// TIA Portal V19 program export: 1 tag tables, 0 data types, 14 data blocks, 15 code blocks (in call order from the OBs), 30 instance data blocks

VAR_GLOBAL   // PLC tag table "Default tag table"
   "EMG STOP" AT %I0.0 : Bool;
   "HOOTER RESET" AT %I0.1 : Bool;
   "PHASE FAIL" AT %I0.2 : Bool;
   "AIR PRESSURE FAIL" AT %I0.3 : Bool;
   "SYRUP MFG VESSEL BOTTOM STERROR TRIP" AT %I0.4 : Bool;
   "PREMIXING VESSEL BOTTOM STERROR TRIP" AT %I0.5 : Bool;
   "INLINE 1 HOMOGENIZER MOTOR1 TRIP" AT %I0.6 : Bool;
   "INLINE 2 HOMOGENIZER MOTOR 2 TRIP" AT %I0.7 : Bool;
   "FILTER PRESS MOTOR 1 TRIP" AT %I1.0 : Bool;
   "FILTER PRESS MOTOR 2 TRIP" AT %I1.1 : Bool;
   "VACCUM PUMP MOTOR 1 TRIP" AT %I1.2 : Bool;
   "VACCUMP PUMP MOTOR 2 TRIP" AT %I1.3 : Bool;
   "VACCUMP PUMP MOTOR 3 TRIP" AT %I1.4 : Bool;
   "VACCUMP PUMP MOTOR 4 TRIP" AT %I1.5 : Bool;
   "SUGAR VESSEL BOTTOM STERROR TRIP" AT %I1.6 : Bool;
   "BASKET FILTER MOTOR TRIP" AT %I1.7 : Bool;
   "SYRUP FLOW SWITCH" AT %I2.0 : Bool;
   "PREMIXING FLOW SWITCH" AT %I2.1 : Bool;
   "SUGAR FLOW SWITCH" AT %I2.2 : Bool;
   "INLINE 1 FLOW SWITCH" AT %I2.3 : Bool;
   "INLINE 2 FLOW SWITCH" AT %I2.4 : Bool;
   "HOOTER RESET 2" AT %I2.5 : Bool;
   SPARE_DI1 AT %I2.6 : Bool;
   SPARE_DI2 AT %I2.7 : Bool;
   SPARE_DI3 AT %I3.0 : Bool;
   SPARE_DI4 AT %I3.1 : Bool;
   SPARE_DI5 AT %I3.2 : Bool;
   SPARE_DI6 AT %I3.3 : Bool;
   SPARE_DI7 AT %I3.4 : Bool;
   SPARE_DI8 AT %I3.5 : Bool;
   SPARE_DI9 AT %I3.6 : Bool;
   SPARE_DI10 AT %I3.7 : Bool;
   "SYRUP MFG VESSEL BOTTOM STERROR RUN" AT %Q0.0 : Bool;
   "PREMIXING VESSEL BOTTOM STERROR RUN" AT %Q0.1 : Bool;
   "INLINE 1 HOMOGENIZER MOTOR1 RUN" AT %Q0.2 : Bool;
   "INLINE 2 HOMOGENIZER MOTOR 2 RUN" AT %Q0.3 : Bool;
   "FILTER PRESS MOTOR 1 RUN" AT %Q0.4 : Bool;
   "FILTER PRESS MOTOR 2 RUN" AT %Q0.5 : Bool;
   "VACCUM PUMP MOTOR 1 RUN" AT %Q0.6 : Bool;
   "VACCUMP PUMP MOTOR 2 RUN" AT %Q0.7 : Bool;
   "VACCUMP PUMP MOTOR 3 RUN" AT %Q1.0 : Bool;
   "VACCUMP PUMP MOTOR 4 RUN" AT %Q1.1 : Bool;
   "SUGAR VESSEL BOTTOM STERROR RUN" AT %Q1.2 : Bool;
   "BASKET FILTER MOTOR RUN" AT %Q1.3 : Bool;
   "PBV-01" AT %Q1.4 : Bool;
   "PBV-02" AT %Q1.5 : Bool;
   "PBV-03" AT %Q1.6 : Bool;
   "PBV-04" AT %Q1.7 : Bool;
   "PBV-07" AT %Q2.0 : Bool;
   "PAV-09" AT %Q2.1 : Bool;
   "PAV-10" AT %Q2.2 : Bool;
   "PAV-11" AT %Q2.3 : Bool;
   "PAV-12" AT %Q2.4 : Bool;
   "PAV-13" AT %Q2.5 : Bool;
   "PAV-14" AT %Q2.6 : Bool;
   "PBV-15" AT %Q2.7 : Bool;
   "PBV-16" AT %Q3.0 : Bool;
   "PFBV-17" AT %Q3.1 : Bool;
   "PBV-19" AT %Q3.2 : Bool;
   "PBV-20" AT %Q3.3 : Bool;
   "PBV-21" AT %Q3.4 : Bool;
   "PBV-22" AT %Q3.5 : Bool;
   "PBV-25" AT %Q3.6 : Bool;
   "PBV-27" AT %Q3.7 : Bool;
   "PAV-28" AT %Q4.0 : Bool;
   "PAV-29" AT %Q4.1 : Bool;
   "PBV-30" AT %Q4.2 : Bool;
   "PBV-31" AT %Q4.3 : Bool;
   "PFBV-32" AT %Q4.4 : Bool;
   "PBV-36" AT %Q4.5 : Bool;
   "PBV-37" AT %Q4.6 : Bool;
   "PBV-38" AT %Q4.7 : Bool;
   "PBV-41" AT %Q5.0 : Bool;
   "PAV-50" AT %Q5.1 : Bool;
   "PAV-51" AT %Q5.2 : Bool;
   "PAV-52" AT %Q5.3 : Bool;
   "PAV-53" AT %Q5.4 : Bool;
   "PAV-54" AT %Q5.5 : Bool;
   "PAV-55" AT %Q5.6 : Bool;
   "PAV-56" AT %Q5.7 : Bool;
   "PBV-57" AT %Q6.0 : Bool;
   "PFBV-59" AT %Q6.1 : Bool;
   "PBV-79" AT %Q6.2 : Bool;
   "PBV-80" AT %Q6.3 : Bool;
   "PBV-81" AT %Q6.4 : Bool;
   "PBV-82" AT %Q6.5 : Bool;
   "PBV-83" AT %Q6.6 : Bool;
   "PBV-84" AT %Q6.7 : Bool;
   "PBV-85" AT %Q7.0 : Bool;
   "PBV-86" AT %Q7.1 : Bool;
   "PBV-87" AT %Q7.2 : Bool;
   "PBV-88" AT %Q7.3 : Bool;
   "PBV-89" AT %Q7.4 : Bool;
   "PBV-90" AT %Q7.5 : Bool;
   "PBV-91" AT %Q7.6 : Bool;
   "PBV-92" AT %Q7.7 : Bool;
   "PBV-93" AT %Q8.0 : Bool;
   "PBV-94" AT %Q8.1 : Bool;
   "PBV-95" AT %Q8.2 : Bool;
   "PBV-96" AT %Q8.3 : Bool;
   "PBV-97" AT %Q8.4 : Bool;
   "PBV-98" AT %Q8.5 : Bool;
   "PAV-99" AT %Q8.6 : Bool;
   "PBV-100" AT %Q8.7 : Bool;
   "PBV-101" AT %Q9.0 : Bool;
   "PBV-102" AT %Q9.1 : Bool;
   "PBV-103" AT %Q9.2 : Bool;
   "PBV-104" AT %Q9.3 : Bool;
   "PBV-105" AT %Q9.4 : Bool;
   "PBV-106" AT %Q9.5 : Bool;
   "PBV-107" AT %Q9.6 : Bool;
   "PBV-108" AT %Q9.7 : Bool;
   "PBV-109" AT %Q10.0 : Bool;
   "PBV-110" AT %Q10.1 : Bool;
   "PBV-111" AT %Q10.2 : Bool;
   "PBV-112" AT %Q10.3 : Bool;
   "PAV-113" AT %Q10.4 : Bool;
   "PBV-114" AT %Q10.5 : Bool;
   "PBV-115" AT %Q10.6 : Bool;
   "PBV-116" AT %Q10.7 : Bool;
   "PBV-117" AT %Q11.0 : Bool;
   "PBV-118" AT %Q11.1 : Bool;
   "PBV-119" AT %Q11.2 : Bool;
   "PBV-120" AT %Q11.3 : Bool;
   "PBV-121" AT %Q11.4 : Bool;
   "PBV-122" AT %Q11.5 : Bool;
   "PBV-123" AT %Q11.6 : Bool;
   "PBV-124" AT %Q11.7 : Bool;
   "PBV-149" AT %Q12.0 : Bool;
   "PBV-150" AT %Q12.1 : Bool;
   "PBV-151" AT %Q12.2 : Bool;
   "PBV-152" AT %Q12.3 : Bool;
   "PBV-153" AT %Q12.4 : Bool;
   "PBV-155" AT %Q12.5 : Bool;
   "PBV-156" AT %Q12.6 : Bool;
   HOOTER_1 AT %Q12.7 : Bool;
   HOOTR_2 AT %Q13.0 : Bool;
   SPARE_DO1 AT %Q13.1 : Bool;
   SPARE_DO2 AT %Q13.2 : Bool;
   SPARE_DO3 AT %Q13.3 : Bool;
   SPARE_DO4 AT %Q13.4 : Bool;
   SPARE_DO5 AT %Q13.5 : Bool;
   SPARE_DO6 AT %Q13.6 : Bool;
   SPARE_DO7 AT %Q13.7 : Bool;
   SPARE_8 AT %Q23.0 : Bool;
   SPARE_9 AT %Q23.1 : Bool;
   SPARE_10 AT %Q23.2 : Bool;
   SPARE_11 AT %Q23.3 : Bool;
   SPARE_12 AT %Q23.4 : Bool;
   SPARE_13 AT %Q23.5 : Bool;
   SPARE_14 AT %Q23.6 : Bool;
   SPARE_15 AT %Q23.7 : Bool;
   SPARE_16 AT %Q24.0 : Bool;
   SPARE_17 AT %Q24.1 : Bool;
   SPARE_18 AT %Q24.2 : Bool;
   SPARE_19 AT %Q24.3 : Bool;
   SPARE_20 AT %Q24.4 : Bool;
   SPARE_21 AT %Q24.5 : Bool;
   SPARE_22 AT %Q24.6 : Bool;
   SPARE_23 AT %Q24.7 : Bool;
   "SYRUP VESSEL TEMP SENSOR" AT %IW4 : Int;
   "PREMIXING VESSEL TEMP SENSOR" AT %IW6 : Int;
   "SUGAR VESSEL TEMP SENSOR" AT %IW8 : Int;
   "STEAM LINE_1 TEMP SENSOR" AT %IW10 : Int;
   "STEAM LINE_2 TEMP SENSOR" AT %IW12 : Int;
   "PRESSURE TRANSMITTER 1" AT %IW14 : Int;
   "PRESSURE TRANSMITTER 2" AT %IW16 : Int;
   "VACCIM TRANSMITTER 1" AT %IW18 : Int;
   "VACCIM TRANSMITTER 2" AT %IW20 : Int;
   "VACCUM TRANSMITTER 3" AT %IW22 : Int;
   "SYRUP LOAD CELL" AT %IW24 : Int;
   "PREMIXING LOAD CELL" AT %IW26 : Int;
   "SUGAR LOAD CELL" AT %IW28 : Int;
   "ULTRASONIC LEVEL SENSOR-1" AT %IW30 : Int;
   "ULTRASONIC LEVEL SENSOR-2" AT %IW32 : Int;
   "ULTRASONIC LEVEL SENSOR-3" AT %IW34 : Int;
   "SYRUP MFG VESSEL SPEED" AT %QW15 : Int;
   "PREMIXING VESSEL SPEED" AT %QW17 : Int;
   "SUGAR VESSEL SPEED" AT %QW19 : Int;
   "SPARE(17)" AT %QW21 : Int;
   System_Byte AT %MB1 : Byte;
   DiagStatusUpdate AT %M1.1 : Bool;
   AlwaysTRUE AT %M1.2 : Bool;
   AlwaysFALSE AT %M1.3 : Bool;
   Clock_Byte AT %MB0 : Byte;
   Clock_10Hz AT %M0.0 : Bool;
   Clock_5Hz AT %M0.1 : Bool;
   "Clock_2.5Hz" AT %M0.2 : Bool;
   Clock_2Hz AT %M0.3 : Bool;
   "Clock_1.25Hz" AT %M0.4 : Bool;
   Clock_1Hz AT %M0.5 : Bool;
   "Clock_0.625Hz" AT %M0.6 : Bool;
   "Clock_0.5Hz" AT %M0.7 : Bool;
   "Vaccup Pump2-W bit" AT %M6.0 : Bool;
   "Vaccup Pump2-S bit" AT %M6.1 : Bool;
   YY AT %M4.0 : Bool;
   "MFG LOVE CALCULATE PV" AT %MD8 : Real;
   hh1 AT %MD12 : Real;
   "MFG MOVE PV LOAD CELL" AT %MD16 : Real;
   LL AT %M2.0 : Bool;
END_VAR

DATA_BLOCK "DI MAPING"   // DB1
{ S7_Optimized_Access := 'FALSE' }
   VAR
      "EMG STOP" : Bool;
      "HOOTER RESET_1" : Bool;
      "PHASE FAIL" : Bool;
      "AIR PRESSURE FAIL" : Bool;
      "SYRUP MFG VESSEL BOTTOM STERROR TRIP" : Bool;
      "PREMIXING VESSEL BOTTOM STERROR TRIP" : Bool;
      "INLINE 1 HOMOGENIZER MOTOR1 TRIP" : Bool;
      "INLINE 2 HOMOGENIZER MOTOR 2 TRIP" : Bool;
      "FILTER PRESS MOTOR 1 TRIP" : Bool;
      "FILTER PRESS MOTOR 2 TRIP" : Bool;
      "VACCUM PUMP MOTOR 1 TRIP" : Bool;
      "VACCUMP PUMP MOTOR 2 TRIP" : Bool;
      "VACCUMP PUMP MOTOR 3 TRIP" : Bool;
      "VACCUMP PUMP MOTOR 4 TRIP" : Bool;
      "SUGAR VESSEL BOTTOM STERROR TRIP" : Bool;
      "BASKET FILTER MOTOR TRIP" : Bool;
      "SYRUP FLOW SWITCH" : Bool;
      "PREMIXING FLOW SWITCH" : Bool;
      "SUGAR FLOW SWITCH" : Bool;
      "INLINE 1 FLOW SWITCH" : Bool;
      "INLINE 2 FLOW SWITCH" : Bool;
      "HOOTER RESET_2" : Bool;
      SPARE_DI1 : Bool;
      SPARE_DI2 : Bool;
      SPARE_DI3 : Bool;
      SPARE_DI4 : Bool;
      SPARE_DI5 : Bool;
      SPARE_DI6 : Bool;
      SPARE_DI7 : Bool;
      SPARE_DI8 : Bool;
      SPARE_DI9 : Bool;
      SPARE_DI10 : Bool;
   END_VAR
BEGIN
END_DATA_BLOCK

DATA_BLOCK "AUTO SUBOUTPUT DB"   // DB46
{ S7_Optimized_Access := 'TRUE' }
// stored: MemoryReserve 100
   VAR
      "SYRUP MFG VESSEL BOTTOM STERROR RUN" : Bool;
      "PREMIXING VESSEL BOTTOM STERROR RUN" : Bool;
      "INLINE 1 HOMOGENIZER MOTOR1 RUN" : Bool;
      "INLINE 2 HOMOGENIZER MOTOR 2 RUN" : Bool;
      "FILTER PRESS MOTOR 1 RUN" : Bool;
      "FILTER PRESS MOTOR 2 RUN" : Bool;
      "VACCUM PUMP MOTOR-W 1 RUN" : Bool;
      "VACCUMP PUMP MOTOR-S2 RUN" : Bool;
      "VACCUMP PUMP MOTOR-W 3 RUN" : Bool;
      "VACCUMP PUMP MOTOR-S 4 RUN" : Bool;
      "SUGAR VESSEL BOTTOM STERROR RUN" : Bool;
      "BASKET FILTER MOTOR RUN" : Bool;
      "PBV-01 INGREDIENT INLET" : Bool;
      "PBV-02 CIP INLET (SPRAY BALL)" : Bool;
      "PBV-03 VENT FILTER ISOLATION" : Bool;
      "PBV-04 PW INLET" : Bool;
      "PBV-07 PREMIX TANK DRAIN VALVE" : Bool;
      "PAV-09 JACKET STEAM INLET" : Bool;
      "PAV-10 JACKET CONDENSATE DRAIN" : Bool;
      "PAV-11 JACKET BYPASS DRAIN VALVE" : Bool;
      "PAV-12 SEAL COOLING INLET" : Bool;
      "PAV-13 WATER COOLING INLET" : Bool;
      "PAV-14 WATER COOLING OUTLET" : Bool;
      "PBV-15 VACUUM INLET" : Bool;
      "PBV-16 VACUUM VENT VALVE" : Bool;
      "PFBV-17 TANK OUTLET VALVE" : Bool;
      "PBV-19 PW INLET" : Bool;
      "PBV-20 CIP INLET (SPRAY BALL)" : Bool;
      "PBV-21 VENT FILTER ISOLATION" : Bool;
      "PBV-22 INGREDIENT INLET (SUGAR INLET)" : Bool;
      "PBV-25 BOTTOM OUTLET TO DRAIN VALVE" : Bool;
      "PAV-27 JACKET STEAM INLET" : Bool;
      "PAV-28 SEAL COOLING INLET" : Bool;
      "PAV-29 JACKET CONDENSATE DRAIN" : Bool;
      "PBV-30 VACUUM INLET VALVE" : Bool;
      "PBV-31 VACUUM VENT VALVE" : Bool;
      "PFBV-32 TANK OUTLET VALVE" : Bool;
      "PBV-36 PW INLET" : Bool;
      "PBV-37 VENT FILTER ISOLATION" : Bool;
      "PBV-38 CIP INLET LINE" : Bool;
      "PBV-41 MFG TANK DRAIN VALVE" : Bool;
      "PAV-50 JACKET STEAM INLET" : Bool;
      "PAV-51 WATER COOLING OUTLET" : Bool;
      "PAV-52 WATER COOLING INLET" : Bool;
      "PAV-53 SEAL COOLING INLET" : Bool;
      "PAV-54 JACKET STEAM OUTLET VALVE" : Bool;
      "PAV-55 JACKET CONDENSATE BYPASS DRAIN" : Bool;
      "PAV-56 INLINE HOMO. SEAL COOLING INLET" : Bool;
      "PBV-57 VACUUM INLET VALVE" : Bool;
      "PFBV-59 TANK OUTLET VALVE" : Bool;
      "PBV-79 BASKET FILTER INLET" : Bool;
      "PBV-80 BOTTOM OUTLET TO BASKET FILTER" : Bool;
      "PBV-81 TANK BOTTOM OUTLET TO CIP OUTLET" : Bool;
      "PBV-82 CIP ISOLATION" : Bool;
      "PBV-83 PREMIX TRANSFER TO MFG VESSEL TRANSFER (TOP DISH)" : Bool;
      "PBV-84 FROM TANK OUTLET TO CIP OUTLET" : Bool;
      "PBV-85 SORBITOL INLET LINE" : Bool;
      "PBV-86 GLUCOSE INLET LINE" : Bool;
      "PBV-87 BASKET FILTER TO PREMIX VESSEL LINE" : Bool;
      "PBV-88 BASKET FILTER TRANSFER LINE" : Bool;
      "PBV-89 BASKET FILTER TO MFG INLET TRANSFER LINE" : Bool;
      "PBV-90 PREMIX TO MFG TRANSFER LINE" : Bool;
      "PBV-91 PREMIX TO MFG TRANSFER LINE" : Bool;
      "PBV-92 PREMIX TO STORAGE – 4 TRANSFER LINE" : Bool;
      "PBV-93 TANK OUTLET TO INLINE HOMOGENIZER LINE" : Bool;
      "PBV-94 INLINE HOMOGENIZER INLET LINE" : Bool;
      "PBV-95 TANK OUTLET TO FILTER PRESS LINE" : Bool;
      "PBV-96 INLINE HOMOGENIZER RECIRCULATION LINE" : Bool;
      "PBV-97 FILTER PRESS OUTLET" : Bool;
      "PBV-98 INLINE HOMOGENIZER TO FILTER PRESS OUTLET LINE" : Bool;
      "PAV-99 INLINE HOMOGENIZER SEAL COOLING" : Bool;
      "PBV-100 FILTER PRESS INLET" : Bool;
      "PBV-101 SUGAR MELTING TO MFG TRANSFER (TOP DISH)" : Bool;
      "PBV-102 PREMIX TO MFG TRANSFER (TOP DISH)" : Bool;
      "PBV-103 CIP INLET (SPRAY BALL)" : Bool;
      "PBV-104 MFG VESSEL TRANSFER LINE" : Bool;
      "PBV-105 INGREDIENT INLET" : Bool;
      "PBV-106 SORBITOL INLET" : Bool;
      "PBV-107 GLUCOSE INLET" : Bool;
      "PBV-108 INLINE HOMOGENIZER TO FILTER PRESS INLET LINE" : Bool;
      "PBV-109 HOMO. RECIRCULATION INLET" : Bool;
      "PBV-110 INLINE HOMOGENIZER TO INLET LINE" : Bool;
      "PBV-111 FILTER PRESS OUTLER VALVE" : Bool;
      "PBV-112 FILTER PRESS TO TRANSFER LINE" : Bool;
      "PAV-113 TANK OUTLET TO CIP DRAIN LINE" : Bool;
      "PBV-114 TANK OUTLET TO INLINE HOMOGENIZER LINE" : Bool;
      "PBV-115 MFG TO STORAGE – 1 TRANSFER LINE" : Bool;
      "PBV-116 MFG TO STORAGE – 2 TRANSFER LINE" : Bool;
      "PBV-117 MFG TO STORAGE – 3 TRANSFER LINE" : Bool;
      "PBV-118 FILTER PRESS INLET" : Bool;
      "PBV-119 SEAL COOLING FOR STORAGE VESSEL - 4" : Bool;
      "PBV-120 SEAL COOLING FOR STORAGE VESSEL - 3" : Bool;
      "PBV-121 SEAL COOLING FOR STORAGE VESSEL - 2" : Bool;
      "PBV-122 SEAL COOLING FOR STORAGE VESSEL - 1" : Bool;
      "PBV-123 VESSEL TOP DISH" : Bool;
      "PBV-124 VESSEL INLET LINE" : Bool;
      "PBV-149" : Bool;
      "PBV-150" : Bool;
      "PBV-151" : Bool;
      "PBV-152" : Bool;
      "PBV-153" : Bool;
      "PBV-155" : Bool;
      "PBV-156" : Bool;
   END_VAR
BEGIN
END_DATA_BLOCK

DATA_BLOCK "MANUAL BIT"   // DB4
{ S7_Optimized_Access := 'TRUE' }
// stored: MemoryReserve 100
   VAR
      "SYRUP MFG VESSEL BOTTOM STERROR RUN" : Bool;
      "PREMIXING VESSEL BOTTOM STERROR RUN" : Bool;
      "INLINE 1 HOMOGENIZER MOTOR1 RUN" : Bool;
      "INLINE 2 HOMOGENIZER MOTOR 2 RUN" : Bool;
      "FILTER PRESS MOTOR 1 RUN" : Bool;
      "FILTER PRESS MOTOR 2 RUN" : Bool;
      "VACCUM PUMP MOTOR-W 1 RUN" : Bool;
      "VACCUMP PUMP MOTOR-S2 RUN" : Bool;
      "VACCUM PUMP MOTOR-W 1 RUN_1" : Bool;
      "VACCUMP PUMP MOTOR-S2 RUN_1" : Bool;
      "VACCUMP PUMP MOTOR-W 3 RUN" : Bool;
      "VACCUMP PUMP MOTOR-S 4 RUN" : Bool;
      "SUGAR VESSEL BOTTOM STERROR RUN" : Bool;
      "BASKET FILTER MOTOR RUN" : Bool;
      "PBV-01 INGREDIENT INLET" : Bool;
      "PBV-02 CIP INLET (SPRAY BALL)" : Bool;
      "PBV-03 VENT FILTER ISOLATION" : Bool;
      "PBV-04 PW INLET" : Bool;
      "PBV-07 PREMIX TANK DRAIN VALVE" : Bool;
      "PAV-09 JACKET STEAM INLET" : Bool;
      "PAV-10 JACKET CONDENSATE DRAIN" : Bool;
      "PAV-11 JACKET BYPASS DRAIN VALVE" : Bool;
      "PAV-12 SEAL COOLING INLET" : Bool;
      "PAV-13 WATER COOLING INLET" : Bool;
      "PAV-14 WATER COOLING OUTLET" : Bool;
      "PBV-15 VACUUM INLET" : Bool;
      "PBV-16 VACUUM VENT VALVE" : Bool;
      "PFBV-17 TANK OUTLET VALVE" : Bool;
      "PBV-19 PW INLET" : Bool;
      "PBV-20 CIP INLET (SPRAY BALL)" : Bool;
      "PBV-21 VENT FILTER ISOLATION" : Bool;
      "PBV-22 INGREDIENT INLET (SUGAR INLET)" : Bool;
      "PBV-25 BOTTOM OUTLET TO DRAIN VALVE" : Bool;
      "PAV-27 JACKET STEAM INLET" : Bool;
      "PAV-28 SEAL COOLING INLET" : Bool;
      "PAV-29 JACKET CONDENSATE DRAIN" : Bool;
      "PBV-30 VACUUM INLET VALVE" : Bool;
      "PBV-31 VACUUM VENT VALVE" : Bool;
      "PFBV-32 TANK OUTLET VALVE" : Bool;
      "PBV-36 PW INLET" : Bool;
      "PBV-37 VENT FILTER ISOLATION" : Bool;
      "PBV-38 CIP INLET LINE" : Bool;
      "PBV-41 MFG TANK DRAIN VALVE" : Bool;
      "PAV-50 JACKET STEAM INLET" : Bool;
      "PAV-51 WATER COOLING OUTLET" : Bool;
      "PAV-52 WATER COOLING INLET" : Bool;
      "PAV-53 SEAL COOLING INLET" : Bool;
      "PAV-54 JACKET STEAM OUTLET VALVE" : Bool;
      "PAV-55 JACKET CONDENSATE BYPASS DRAIN" : Bool;
      "PAV-56 INLINE HOMO. SEAL COOLING INLET" : Bool;
      "PBV-57 VACUUM INLET VALVE" : Bool;
      "PFBV-59 TANK OUTLET VALVE" : Bool;
      "PBV-79 BASKET FILTER INLET" : Bool;
      "PBV-80 BOTTOM OUTLET TO BASKET FILTER" : Bool;
      "PBV-81 TANK BOTTOM OUTLET TO CIP OUTLET" : Bool;
      "PBV-82 CIP ISOLATION" : Bool;
      "PBV-83 PREMIX TRANSFER TO MFG VESSEL TRANSFER (TOP DISH)" : Bool;
      "PBV-84 FROM TANK OUTLET TO CIP OUTLET" : Bool;
      "PBV-85 SORBITOL INLET LINE" : Bool;
      "PBV-86 GLUCOSE INLET LINE" : Bool;
      "PBV-87 BASKET FILTER TO PREMIX VESSEL LINE" : Bool;
      "PBV-88 BASKET FILTER TRANSFER LINE" : Bool;
      "PBV-89 BASKET FILTER TO MFG INLET TRANSFER LINE" : Bool;
      "PBV-90 PREMIX TO MFG TRANSFER LINE" : Bool;
      "PBV-91 PREMIX TO MFG TRANSFER LINE" : Bool;
      "PBV-92 PREMIX TO STORAGE – 4 TRANSFER LINE" : Bool;
      "PBV-93 TANK OUTLET TO INLINE HOMOGENIZER LINE" : Bool;
      "PBV-94 INLINE HOMOGENIZER INLET LINE" : Bool;
      "PBV-95 TANK OUTLET TO FILTER PRESS LINE" : Bool;
      "PBV-96 INLINE HOMOGENIZER RECIRCULATION LINE" : Bool;
      "PBV-97 FILTER PRESS OUTLET" : Bool;
      "PBV-98 INLINE HOMOGENIZER TO FILTER PRESS OUTLET LINE" : Bool;
      "PAV-99 INLINE HOMOGENIZER SEAL COOLING" : Bool;
      "PBV-100 FILTER PRESS INLET" : Bool;
      "PBV-101 SUGAR MELTING TO MFG TRANSFER (TOP DISH)" : Bool;
      "PBV-102 PREMIX TO MFG TRANSFER (TOP DISH)" : Bool;
      "PBV-103 CIP INLET (SPRAY BALL)" : Bool;
      "PBV-104 MFG VESSEL TRANSFER LINE" : Bool;
      "PBV-105 INGREDIENT INLET" : Bool;
      "PBV-106 SORBITOL INLET" : Bool;
      "PBV-107 GLUCOSE INLET" : Bool;
      "PBV-108 INLINE HOMOGENIZER TO FILTER PRESS INLET LINE" : Bool;
      "PBV-109 HOMO. RECIRCULATION INLET" : Bool;
      "PBV-110 INLINE HOMOGENIZER TO INLET LINE" : Bool;
      "PBV-111 FILTER PRESS OUTLER VALVE" : Bool;
      "PBV-112 FILTER PRESS TO TRANSFER LINE" : Bool;
      "PAV-113 TANK OUTLET TO CIP DRAIN LINE" : Bool;
      "PBV-114 TANK OUTLET TO INLINE HOMOGENIZER LINE" : Bool;
      "PBV-115 MFG TO STORAGE – 1 TRANSFER LINE" : Bool;
      "PBV-116 MFG TO STORAGE – 2 TRANSFER LINE" : Bool;
      "PBV-117 MFG TO STORAGE – 3 TRANSFER LINE" : Bool;
      "PBV-118 FILTER PRESS INLET" : Bool;
      "PBV-119 SEAL COOLING FOR STORAGE VESSEL - 4" : Bool;
      "PBV-120 SEAL COOLING FOR STORAGE VESSEL - 3" : Bool;
      "PBV-121 SEAL COOLING FOR STORAGE VESSEL - 2" : Bool;
      "PBV-122 SEAL COOLING FOR STORAGE VESSEL - 1" : Bool;
      "PBV-123 VESSEL TOP DISH" : Bool;
      "PBV-124 VESSEL INLET LINE" : Bool;
      "PBV-149" : Bool;
      "PBV-150" : Bool;
      "PBV-151" : Bool;
      "PBV-152" : Bool;
      "PBV-153" : Bool;
      "PBV-155" : Bool;
      "PBV-156" : Bool;
      HOOTER_1 : Bool;
      HOOTR_2 : Bool;
   END_VAR
BEGIN
END_DATA_BLOCK

DATA_BLOCK "RECIRCULATION DB"   // DB63
{ S7_Optimized_Access := 'TRUE' }
// stored: MemoryReserve 100
   VAR RETAIN
      MFG : Struct
         START : Bool;
         STOP : Bool;
         PAUSE : Bool;
         BUFF : Int;
      END_STRUCT;
      PREMIXING : Struct
         START : Bool;
         STOP : Bool;
         PAUSE : Bool;
         BUFF : Int;
      END_STRUCT;
      "MFG RECIRCULATION TIME SET" : Int;
   END_VAR
   VAR
      "MFG RECIRCULATION TIME PV" : Int;
   END_VAR
   VAR RETAIN
      "PREMIXING RECIRCULATION TIME SET" : Int;
   END_VAR
   VAR
      "PREMIXING RECIRCULATION TIME PV" : Int;
   END_VAR
BEGIN
END_DATA_BLOCK

DATA_BLOCK "TRANSFER DB"   // DB15
{ S7_Optimized_Access := 'TRUE' }
// stored: MemoryReserve 100
   VAR
      "MFG VACCUM PUMP MOTOR-W 1 BIT" : Bool;
      "MFG VACCUMP PUMP MOTOR-S2 BIT" : Bool;
      "PREMIXING VACCUM PUMP MOTOR-W 1 BIT" : Bool;
      "PREMIXING VACCUMP PUMP MOTOR-S2 BIT" : Bool;
      "SUAGR VACCUM PUMP MOTOR-W 3 BIT" : Bool;
      "SUGAR VACCUMP PUMP MOTOR-S4 BIT" : Bool;
      START : Struct
         "SUGAR TO PREMIXING" : Bool;
         "SUGAR TO MFG" : Bool;
         "PREMIXING TO MFG WITH INLINE HOMO" : Bool;
         "PREMIXING TO MFG WITH INLINE FILTER PRES" : Bool;
         "PREMIXING TO STORAGE-4 WITH INLINE HOMO" : Bool;
         "PREMIXING TO STORAGE-4 WITH INLINE FILTER PRES" : Bool;
         "MFG TO STORAGE-1 WITH INLINE HOMO" : Bool;
         "MFG TO STORAGE-1 WITH INLINE FILTER PRES" : Bool;
         "MFG TO STORAGE-2 WITH INLINE HOMO" : Bool;
         "MFG TO STORAGE-2 WITH INLINE FILTER PRES" : Bool;
         "MFG TO STORAGE-3 WITH INLINE HOMO" : Bool;
         "MFG TO STORAGE-3 WITH INLINE FILTER PRES" : Bool;
      END_STRUCT;
      STOP : Struct
         "SUGAR TO PREMIXING" : Bool;
         "SUGAR TO MFG" : Bool;
         "PREMIXING TO MFG WITH INLINE HOMO" : Bool;
         "PREMIXING TO MFG WITH INLINE FILTER PRES" : Bool;
         "PREMIXING TO STORAGE-4 WITH INLINE HOMO" : Bool;
         "PREMIXING TO STORAGE-4 WITH INLINE FILTER PRES" : Bool;
         "MFG TO STORAGE-1 WITH INLINE HOMO" : Bool;
         "MFG TO STORAGE-1 WITH INLINE FILTER PRES" : Bool;
         "MFG TO STORAGE-2 WITH INLINE HOMO" : Bool;
         "MFG TO STORAGE-2 WITH INLINE FILTER PRES" : Bool;
         "MFG TO STORAGE-3 WITH INLINE HOMO" : Bool;
         "MFG TO STORAGE-3 WITH INLINE FILTER PRES" : Bool;
      END_STRUCT;
   END_VAR
   VAR RETAIN
      PAUSE : Struct
         "SUGAR TO PREMIXING" : Bool;
         "SUGAR TO MFG" : Bool;
         "PREMIXING TO MFG WITH INLINE HOMO" : Bool;
         "PREMIXING TO MFG WITH INLINE FILTER PRES" : Bool;
         "PREMIXING TO STORAGE-4 WITH INLINE HOMO" : Bool;
         "PREMIXING TO STORAGE-4 WITH INLINE FILTER PRES" : Bool;
         "MFG TO STORAGE-1 WITH INLINE HOMO" : Bool;
         "MFG TO STORAGE-1 WITH INLINE FILTER PRES" : Bool;
         "MFG TO STORAGE-2 WITH INLINE HOMO" : Bool;
         "MFG TO STORAGE-2 WITH INLINE FILTER PRES" : Bool;
         "MFG TO STORAGE-3 WITH INLINE HOMO" : Bool;
         "MFG TO STORAGE-3 WITH INLINE FILTER PRES" : Bool;
      END_STRUCT;
      BUFF : Struct
         "SUGAR TO PREMIXING" : Int;
         "SUGAR TO MFG" : Int;
         "PREMIXING TO MFG WITH INLINE HOMO" : Int;
         "PREMIXING TO MFG WITH INLINE FILTER PRES" : Int;
         "PREMIXING TO STORAGE-4 WITH INLINE HOMO" : Int;
         "PREMIXING TO STORAGE-4 WITH INLINE FILTER PRES" : Int;
         "MFG TO STORAGE-1 WITH INLINE HOMO" : Int;
         "MFG TO STORAGE-1 WITH INLINE FILTER PRES" : Int;
         "MFG TO STORAGE-2 WITH INLINE HOMO" : Int;
         "MFG TO STORAGE-2 WITH INLINE FILTER PRES" : Int;
         "MFG TO STORAGE-3 WITH INLINE HOMO" : Int;
         "MFG TO STORAGE-3 WITH INLINE FILTER PRES" : Int;
      END_STRUCT;
   END_VAR
   VAR
      BIT : Struct
         "SUGAR TO PREMIXING" : Struct
            "PFBV-32 TANK OUTLET VALVE" : Bool;
            "PBV-80 BOTTOM OUTLET TO BASKET FILTER" : Bool;
            "BASKET FILTER MOTOR RUN" : Bool;
            "PBV-79 BASKET FILTER INLET" : Bool;
            "PBV-149" : Bool;
            "PBV-88 BASKET FILTER TRANSFER LINE" : Bool;
            "PBV-87 BASKET FILTER TO PREMIX VESSEL LINE" : Bool;
         END_STRUCT;
         "SUGAR TO MFG" : Struct
            "PFBV-32 TANK OUTLET VALVE" : Bool;
            "PBV-80 BOTTOM OUTLET TO BASKET FILTER" : Bool;
            "BASKET FILTER MOTOR RUN" : Bool;
            "PBV-79 BASKET FILTER INLET" : Bool;
            "PBV-149" : Bool;
            "PBV-89 BASKET FILTER TO MFG INLET TRANSFER LINE" : Bool;
            "PBV-101 SUGAR MELTING TO MFG TRANSFER (TOP DISH)" : Bool;
         END_STRUCT;
         "PREMIXING TO MFG WITH INLINE HOMO" : Struct
            "PFBV-17 TANK OUTLET VALVE" : Bool;
            "PBV-93 TANK OUTLET TO INLINE HOMOGENIZER LINE" : Bool;
            "PBV-94 INLINE HOMOGENIZER INLET LINE" : Bool;
            "INLINE 2 HOMOGENIZER MOTOR 2 RUN" : Bool;
            "PBV-96 INLINE HOMOGENIZER RECIRCULATION LINE" : Bool;
            "PBV-91 PREMIX TO MFG TRANSFER LINE" : Bool;
            "PBV-102 PREMIX TO MFG TRANSFER (TOP DISH)" : Bool;
         END_STRUCT;
         "PREMIXING TO MFG WITH INLINE FILTER PRES" : Struct
            "PFBV-17 TANK OUTLET VALVE" : Bool;
            "PBV-93 TANK OUTLET TO INLINE HOMOGENIZER LINE" : Bool;
            "PBV-95 TANK OUTLET TO FILTER PRESS LINE" : Bool;
            "FILTER PRESS MOTOR 2 RUN" : Bool;
            "PBV-100 FILTER PRESS INLET" : Bool;
            "PBV-97 FILTER PRESS OUTLET" : Bool;
            "PBV-98 INLINE HOMOGENIZER TO FILTER PRESS OUTLET LINE" : Bool;
            "PBV-91 PREMIX TO MFG TRANSFER LINE" : Bool;
            "PBV-102 PREMIX TO MFG TRANSFER (TOP DISH)" : Bool;
         END_STRUCT;
         "PREMIXING TO STORAGE-4 WITH INLINE HOMO" : Struct
            "PFBV-17 TANK OUTLET VALVE" : Bool;
            "PBV-93 TANK OUTLET TO INLINE HOMOGENIZER LINE" : Bool;
            "PBV-94 INLINE HOMOGENIZER INLET LINE" : Bool;
            "INLINE 2 HOMOGENIZER MOTOR 2 RUN" : Bool;
            "PBV-96 INLINE HOMOGENIZER RECIRCULATION LINE" : Bool;
            "PBV-92 PREMIX TO STORAGE – 4 TRANSFER LINE" : Bool;
         END_STRUCT;
         "PREMIXING TO STORAGE-4 WITH INLINE FILTER PRES" : Struct
            "PFBV-17 TANK OUTLET VALVE" : Bool;
            "PBV-93 TANK OUTLET TO INLINE HOMOGENIZER LINE" : Bool;
            "PBV-95 TANK OUTLET TO FILTER PRESS LINE" : Bool;
            "FILTER PRESS MOTOR 2 RUN" : Bool;
            "PBV-100 FILTER PRESS INLET" : Bool;
            "PBV-97 FILTER PRESS OUTLET" : Bool;
            "PBV-98 INLINE HOMOGENIZER TO FILTER PRESS OUTLET LINE" : Bool;
            "PBV-92 PREMIX TO STORAGE – 4 TRANSFER LINE" : Bool;
         END_STRUCT;
         "MFG TO STORAGE-1 WITH INLINE HOMO" : Struct
            "PFBV-59 TANK OUTLET VALVE" : Bool;
            "PBV-114 TANK OUTLET TO INLINE HOMOGENIZER LINE" : Bool;
            "PBV-110 INLINE HOMOGENIZER TO INLET LINE" : Bool;
            "PAV-56 INLINE HOMO. SEAL COOLING INLET" : Bool;
            "INLINE 1 HOMOGENIZER MOTOR1 RUN" : Bool;
            "PBV-109 HOMO. RECIRCULATION INLET" : Bool;
            "PBV-115 MFG TO STORAGE – 1 TRANSFER LINE" : Bool;
         END_STRUCT;
         "MFG TO STORAGE-1 WITH INLINE FILTER PRES" : Struct
            "PFBV-59 TANK OUTLET VALVE" : Bool;
            "PBV-114 TANK OUTLET TO INLINE HOMOGENIZER LINE" : Bool;
            "PBV-108 INLINE HOMOGENIZER TO FILTER PRESS INLET LINE" : Bool;
            "FILTER PRESS MOTOR 1 RUN" : Bool;
            "PBV-118 FILTER PRESS INLET" : Bool;
            "PBV-111 FILTER PRESS OUTLER VALVE" : Bool;
            "PBV-112 FILTER PRESS TO TRANSFER LINE" : Bool;
            "PBV-115 MFG TO STORAGE – 1 TRANSFER LINE" : Bool;
         END_STRUCT;
         "MFG TO STORAGE-2 WITH INLINE HOMO" : Struct
            "PFBV-59 TANK OUTLET VALVE" : Bool;
            "PBV-114 TANK OUTLET TO INLINE HOMOGENIZER LINE" : Bool;
            "PBV-110 INLINE HOMOGENIZER TO INLET LINE" : Bool;
            "PAV-56 INLINE HOMO. SEAL COOLING INLET" : Bool;
            "INLINE 1 HOMOGENIZER MOTOR1 RUN" : Bool;
            "PBV-109 HOMO. RECIRCULATION INLET" : Bool;
            "PBV-116 MFG TO STORAGE – 2 TRANSFER LINE" : Bool;
         END_STRUCT;
         "MFG TO STORAGE-2 WITH INLINE FILTER PRES" : Struct
            "PFBV-59 TANK OUTLET VALVE" : Bool;
            "PBV-114 TANK OUTLET TO INLINE HOMOGENIZER LINE" : Bool;
            "PBV-108 INLINE HOMOGENIZER TO FILTER PRESS INLET LINE" : Bool;
            "FILTER PRESS MOTOR 1 RUN" : Bool;
            "PBV-118 FILTER PRESS INLET" : Bool;
            "PBV-111 FILTER PRESS OUTLER VALVE" : Bool;
            "PBV-112 FILTER PRESS TO TRANSFER LINE" : Bool;
            "PBV-116 MFG TO STORAGE – 2 TRANSFER LINE" : Bool;
         END_STRUCT;
         "MFG TO STORAGE-3 WITH INLINE HOMO" : Struct
            "PFBV-59 TANK OUTLET VALVE" : Bool;
            "PBV-114 TANK OUTLET TO INLINE HOMOGENIZER LINE" : Bool;
            "PBV-110 INLINE HOMOGENIZER TO INLET LINE" : Bool;
            "PAV-56 INLINE HOMO. SEAL COOLING INLET" : Bool;
            "INLINE 1 HOMOGENIZER MOTOR1 RUN" : Bool;
            "PBV-109 HOMO. RECIRCULATION INLET" : Bool;
            "PBV-117 MFG TO STORAGE – 3 TRANSFER LINE" : Bool;
         END_STRUCT;
         "MFG TO STORAGE-3 WITH INLINE FILTER PRES" : Struct
            "PFBV-59 TANK OUTLET VALVE" : Bool;
            "PBV-114 TANK OUTLET TO INLINE HOMOGENIZER LINE" : Bool;
            "PBV-108 INLINE HOMOGENIZER TO FILTER PRESS INLET LINE" : Bool;
            "FILTER PRESS MOTOR 1 RUN" : Bool;
            "PBV-118 FILTER PRESS INLET" : Bool;
            "PBV-111 FILTER PRESS OUTLER VALVE" : Bool;
            "PBV-112 FILTER PRESS TO TRANSFER LINE" : Bool;
            "PBV-117 MFG TO STORAGE – 3 TRANSFER LINE" : Bool;
         END_STRUCT;
      END_STRUCT;
      OUTPUT : Struct
         "SYRUP MFG VESSEL BOTTOM STERROR RUN" : Bool;
         "PREMIXING VESSEL BOTTOM STERROR RUN" : Bool;
         "INLINE 1 HOMOGENIZER MOTOR1 RUN" : Bool;
         "INLINE 2 HOMOGENIZER MOTOR 2 RUN" : Bool;
         "FILTER PRESS MOTOR 1 RUN" : Bool;
         "FILTER PRESS MOTOR 2 RUN" : Bool;
         "VACCUM PUMP MOTOR-W 1 RUN" : Bool;
         "VACCUMP PUMP MOTOR-S2 RUN" : Bool;
         "VACCUMP PUMP MOTOR-W 3 RUN" : Bool;
         "VACCUMP PUMP MOTOR-S 4 RUN" : Bool;
         "SUGAR VESSEL BOTTOM STERROR RUN" : Bool;
         "BASKET FILTER MOTOR RUN" : Bool;
         "PBV-01 INGREDIENT INLET" : Bool;
         "PBV-02 CIP INLET (SPRAY BALL)" : Bool;
         "PBV-03 VENT FILTER ISOLATION" : Bool;
         "PBV-04 PW INLET" : Bool;
         "PBV-07 PREMIX TANK DRAIN VALVE" : Bool;
         "PAV-09 JACKET STEAM INLET" : Bool;
         "PAV-10 JACKET CONDENSATE DRAIN" : Bool;
         "PAV-11 JACKET BYPASS DRAIN VALVE" : Bool;
         "PAV-12 SEAL COOLING INLET" : Bool;
         "PAV-13 WATER COOLING INLET" : Bool;
         "PAV-14 WATER COOLING OUTLET" : Bool;
         "PBV-15 VACUUM INLET" : Bool;
         "PBV-16 VACUUM VENT VALVE" : Bool;
         "PFBV-17 TANK OUTLET VALVE" : Bool;
         "PBV-19 PW INLET" : Bool;
         "PBV-20 CIP INLET (SPRAY BALL)" : Bool;
         "PBV-21 VENT FILTER ISOLATION" : Bool;
         "PBV-22 INGREDIENT INLET (SUGAR INLET)" : Bool;
         "PBV-25 BOTTOM OUTLET TO DRAIN VALVE" : Bool;
         "PAV-27 JACKET STEAM INLET" : Bool;
         "PAV-28 SEAL COOLING INLET" : Bool;
         "PAV-29 JACKET CONDENSATE DRAIN" : Bool;
         "PBV-30 VACUUM INLET VALVE" : Bool;
         "PBV-31 VACUUM VENT VALVE" : Bool;
         "PFBV-32 TANK OUTLET VALVE" : Bool;
         "PBV-36 PW INLET" : Bool;
         "PBV-37 VENT FILTER ISOLATION" : Bool;
         "PBV-38 CIP INLET LINE" : Bool;
         "PBV-41 MFG TANK DRAIN VALVE" : Bool;
         "PAV-50 JACKET STEAM INLET" : Bool;
         "PAV-51 WATER COOLING OUTLET" : Bool;
         "PAV-52 WATER COOLING INLET" : Bool;
         "PAV-53 SEAL COOLING INLET" : Bool;
         "PAV-54 JACKET STEAM OUTLET VALVE" : Bool;
         "PAV-55 JACKET CONDENSATE BYPASS DRAIN" : Bool;
         "PAV-56 INLINE HOMO. SEAL COOLING INLET" : Bool;
         "PBV-57 VACUUM INLET VALVE" : Bool;
         "PFBV-59 TANK OUTLET VALVE" : Bool;
         "PBV-79 BASKET FILTER INLET" : Bool;
         "PBV-80 BOTTOM OUTLET TO BASKET FILTER" : Bool;
         "PBV-81 TANK BOTTOM OUTLET TO CIP OUTLET" : Bool;
         "PBV-82 CIP ISOLATION" : Bool;
         "PBV-83 PREMIX TRANSFER TO MFG VESSEL TRANSFER (TOP DISH)" : Bool;
         "PBV-84 FROM TANK OUTLET TO CIP OUTLET" : Bool;
         "PBV-85 SORBITOL INLET LINE" : Bool;
         "PBV-86 GLUCOSE INLET LINE" : Bool;
         "PBV-87 BASKET FILTER TO PREMIX VESSEL LINE" : Bool;
         "PBV-88 BASKET FILTER TRANSFER LINE" : Bool;
         "PBV-89 BASKET FILTER TO MFG INLET TRANSFER LINE" : Bool;
         "PBV-90 PREMIX TO MFG TRANSFER LINE" : Bool;
         "PBV-91 PREMIX TO MFG TRANSFER LINE" : Bool;
         "PBV-92 PREMIX TO STORAGE – 4 TRANSFER LINE" : Bool;
         "PBV-93 TANK OUTLET TO INLINE HOMOGENIZER LINE" : Bool;
         "PBV-94 INLINE HOMOGENIZER INLET LINE" : Bool;
         "PBV-95 TANK OUTLET TO FILTER PRESS LINE" : Bool;
         "PBV-96 INLINE HOMOGENIZER RECIRCULATION LINE" : Bool;
         "PBV-97 FILTER PRESS OUTLET" : Bool;
         "PBV-98 INLINE HOMOGENIZER TO FILTER PRESS OUTLET LINE" : Bool;
         "PAV-99 INLINE HOMOGENIZER SEAL COOLING" : Bool;
         "PBV-100 FILTER PRESS INLET" : Bool;
         "PBV-101 SUGAR MELTING TO MFG TRANSFER (TOP DISH)" : Bool;
         "PBV-102 PREMIX TO MFG TRANSFER (TOP DISH)" : Bool;
         "PBV-103 CIP INLET (SPRAY BALL)" : Bool;
         "PBV-104 MFG VESSEL TRANSFER LINE" : Bool;
         "PBV-105 INGREDIENT INLET" : Bool;
         "PBV-106 SORBITOL INLET" : Bool;
         "PBV-107 GLUCOSE INLET" : Bool;
         "PBV-108 INLINE HOMOGENIZER TO FILTER PRESS INLET LINE" : Bool;
         "PBV-109 HOMO. RECIRCULATION INLET" : Bool;
         "PBV-110 INLINE HOMOGENIZER TO INLET LINE" : Bool;
         "PBV-111 FILTER PRESS OUTLER VALVE" : Bool;
         "PBV-112 FILTER PRESS TO TRANSFER LINE" : Bool;
         "PAV-113 TANK OUTLET TO CIP DRAIN LINE" : Bool;
         "PBV-114 TANK OUTLET TO INLINE HOMOGENIZER LINE" : Bool;
         "PBV-115 MFG TO STORAGE – 1 TRANSFER LINE" : Bool;
         "PBV-116 MFG TO STORAGE – 2 TRANSFER LINE" : Bool;
         "PBV-117 MFG TO STORAGE – 3 TRANSFER LINE" : Bool;
         "PBV-118 FILTER PRESS INLET" : Bool;
         "PBV-119 SEAL COOLING FOR STORAGE VESSEL - 4" : Bool;
         "PBV-120 SEAL COOLING FOR STORAGE VESSEL - 3" : Bool;
         "PBV-121 SEAL COOLING FOR STORAGE VESSEL - 2" : Bool;
         "PBV-122 SEAL COOLING FOR STORAGE VESSEL - 1" : Bool;
         "PBV-123 VESSEL TOP DISH" : Bool;
         "PBV-124 VESSEL INLET LINE" : Bool;
         "PBV-149" : Bool;
         "PBV-150" : Bool;
         "PBV-151" : Bool;
         "PBV-152" : Bool;
         "PBV-153" : Bool;
         "PBV-155" : Bool;
         "PBV-156" : Bool;
         HOOTER_1 : Bool;
         HOOTR_2 : Bool;
      END_STRUCT;
   END_VAR
BEGIN
END_DATA_BLOCK

DATA_BLOCK "MODE SELECTION DB"   // DB3
{ S7_Optimized_Access := 'TRUE' }
// stored: MemoryReserve 100
   VAR
      STANDBY : Bool;
      AUTO : Bool;
      MANUAL : Bool;
      START : Bool;
      STOP : Bool;
   END_VAR
   VAR RETAIN
      "MODE BUFF" : Int;
      "PROCESS BUFF" : Int;
   END_VAR
BEGIN
END_DATA_BLOCK

DATA_BLOCK "ALARM DB"   // DB9
{ S7_Optimized_Access := 'TRUE' }
// stored: MemoryReserve 100
   VAR
      "EMG STOP" : Bool;
      "PHASE FAIL" : Bool;
      "AIR PRESSURE FAIL" : Bool;
      "SYRUP MFG VESSEL BOTTOM STERROR TRIP" : Bool;
      "PREMIXING VESSEL BOTTOM STERROR TRIP" : Bool;
      "INLINE 1 HOMOGENIZER MOTOR1 TRIP" : Bool;
      "INLINE 2 HOMOGENIZER MOTOR 2 TRIP" : Bool;
      "FILTER PRESS MOTOR 1 TRIP" : Bool;
      "FILTER PRESS MOTOR 2 TRIP" : Bool;
      "VACCUM PUMP MOTOR 1 TRIP" : Bool;
      "VACCUMP PUMP MOTOR 2 TRIP" : Bool;
      "VACCUMP PUMP MOTOR 3 TRIP" : Bool;
      "VACCUMP PUMP MOTOR 4 TRIP" : Bool;
      "SUGAR VESSEL BOTTOM STERROR TRIP" : Bool;
      "BASKET FILTER MOTOR TRIP" : Bool;
      "SYRUP FLOW SWITCH" : Bool;
      "PREMIXING FLOW SWITCH" : Bool;
      "SUGAR FLOW SWITCH" : Bool;
      "INLINE 1 FLOW SWITCH" : Bool;
      "INLINE 2 FLOW SWITCH" : Bool;
      "MFG TO STORAGE-1 WITH INLINE HOMOGENIZER TRANSFER COMPLETE" : Bool;
      "MFG TO STORAGE-1 WITH FILTER PRESS TRANSFER COMPLETE" : Bool;
      "MFG TO STORAGE-2 WITH INLINE HOMOGENIZER TRANSFER COMPLETE" : Bool;
      "MFG TO STORAGE-2 WITH FILTER PRESS TRANSFER COMPLETE" : Bool;
      "MFG TO STORAGE-3 WITH INLINE HOMOGENIZER TRANSFER COMPLETE" : Bool;
      "MFG TO STORAGE-3 WITH FILTER PRESS TRANSFER COMPLETE" : Bool;
      "PREMIXING TRANSFER COMPLETE" : Bool;
      "SUGAR TRANSFER COMPLETE" : Bool;
   END_VAR
BEGIN
END_DATA_BLOCK

DATA_BLOCK "AUTO ALARM DB"   // DB70
{ S7_Optimized_Access := 'TRUE' }
// stored: MemoryReserve 100
   VAR
      "MFG PROCESS" : Struct
         "PURIFIED WATER PROCESS SELECT" : Bool;
         "PURIFIED WATER PROCESS OF INITIAL DRAIN SELECT" : Bool;
         "PURIFIED WATER PROCESS OF LOAD CELL" : Bool;
         "PURIFIED WATER HEATING OR COOLING SELECT" : Bool;
         "PURIFIED WATER PROCESS OF JACKET DRAIN SELECT" : Bool;
         "PURIFIED WATER PROCESS OVER" : Bool;
         "MATERIAL ADDITION PROCESS SELECT" : Bool;
         "MATERIAL ADDITION MATERIAL ADDED TEXT" : Bool;
         "MATERIAL ADDITION DO YOU WANT TO ADD SORBITOL SELECT" : Bool;
         "MATERIAL ADDITION OF SORBITOL OVER" : Bool;
         "MATERIAL ADDITION DO YOU WANT TO ADD GLUCOSE SELECT" : Bool;
         "MATERIAL ADDITION OF GLUCOSE OVER" : Bool;
         "MATERIAL ADDITION PROCESS OVER" : Bool;
         "RECIRCULATION PROCESS SELECT" : Bool;
         "RECIRCULATION PROCESS RUNING" : Bool;
         "RECIRCULATION OVER" : Bool;
         "MFG PROCESS OVER" : Bool;
      END_STRUCT;
      "MFG PROCESS ALARM" : Struct
         "MFG PROCESS START" : Bool;
         "PURIFIED WATER PROCESS START" : Bool;
         "PURIFIED WATER PROCESS OF INITIAL DRAIN START" : Bool;
         "PURIFIED WATER PROCESS OF INITIAL DRAIN STOP" : Bool;
         "PURIFIED WATER PROCESS OF LOAD CELL START" : Bool;
         "PURIFIED WATER PROCESS OF LOAD CELL STOP" : Bool;
         "PURIFIED WATER OF HEATING START" : Bool;
         "PURIFIED WATER OF HEATING STOP" : Bool;
         "PURIFIED WATER OF COOLING START" : Bool;
         "PURIFIED WATER OF COOLING STOP" : Bool;
         "PURIFIED WATER PROCESS OF JACKET DRAIN START" : Bool;
         "PURIFIED WATER PROCESS OF JACKET DRAIN STOP" : Bool;
         "PURIFIED WATER PROCESS OVER" : Bool;
         "MATERIAL ADDITION PROCESS SELECT" : Bool;
         "MATERIAL ADDITION PROCESS START" : Bool;
         "MATERIAL ADDITION OF INITIAL DRAIN SELECT" : Bool;
         "MATERIAL ADDITION OF INITIAL DRAIN START" : Bool;
         "MATERIAL ADDITION OF INITIAL DRAIN STOP" : Bool;
         "MATERIAL ADDITION MATERIAL ADDED TEXT" : Bool;
         "MATERIAL ADDITION DO YOU WANT TO ADD SORBITOL SELECT" : Bool;
         "MATERIAL ADDITION OF SORBITOL START" : Bool;
         "MATERIAL ADDITION OF SORBITOL STIRRER START" : Bool;
         "MATERIAL ADDITION OF SORBITOL STIRRER STOP" : Bool;
         "MATERIAL ADDITION OF SORBITOL OVER" : Bool;
         "MATERIAL ADDITION DO YOU WANT TO ADD GLUCOSE SELECT" : Bool;
         "MATERIAL ADDITION OF GLUCOSE START" : Bool;
         "MATERIAL ADDITION OF GLUCOSE STIRRER START" : Bool;
         "MATERIAL ADDITION OF GLUCOSE STIRRER STOP" : Bool;
         "MATERIAL ADDITION OF GLUCOSE OVER" : Bool;
         "MATERIAL ADDITION PROCESS OF JACKET DRAIN SELECT" : Bool;
         "MATERIAL ADDITION PROCESS OF JACKET DRAIN STOP" : Bool;
         "MATERIAL ADDITION PROCESS OVER" : Bool;
         "RECIRCULATION PROCESS SELECT" : Bool;
         "RECIRCULATION PROCESS START" : Bool;
         "RECIRCULATION PROCESS OF INITIAL DRAIN SELECT" : Bool;
         "RECIRCULATION PROCESS OF INITIAL DRAIN START" : Bool;
         "RECIRCULATION PROCESS OF INITIAL DRAIN STOP" : Bool;
         "RECIRCULATION PROCESS RUNING" : Bool;
         "RECIRCULATION PROCESS OF JACKET DRAIN SELECT" : Bool;
         "RECIRCULATION PROCESS OF JACKET DRAIN STOP" : Bool;
         "RECIRCULATION OVER" : Bool;
         "MFG PROCESS OVER" : Bool;
      END_STRUCT;
      "MFG TRANSFER START" : Struct
         "MFG TO STORAGE-1 WITH INLINE HOMO" : Bool;
         "MFG TO STORAGE-1 WITH INLINE FILTER PRES" : Bool;
         "MFG TO STORAGE-2 WITH INLINE HOMO" : Bool;
         "MFG TO STORAGE-2 WITH INLINE FILTER PRES" : Bool;
         "MFG TO STORAGE-3 WITH INLINE HOMO" : Bool;
         "MFG TO STORAGE-3 WITH INLINE FILTER PRES" : Bool;
      END_STRUCT;
      "MFG TRANSFER OVER" : Struct
         "MFG TO STORAGE-1 WITH INLINE HOMO" : Bool;
         "MFG TO STORAGE-1 WITH INLINE FILTER PRES" : Bool;
         "MFG TO STORAGE-2 WITH INLINE HOMO" : Bool;
         "MFG TO STORAGE-2 WITH INLINE FILTER PRES" : Bool;
         "MFG TO STORAGE-3 WITH INLINE HOMO" : Bool;
         "MFG TO STORAGE-3 WITH INLINE FILTER PRES" : Bool;
      END_STRUCT;
      "MFG MATERIAL SUCTION" : Struct
         "MATERIAL SUCTION START" : Bool;
         "MATERIAL SUCTION OVER" : Bool;
      END_STRUCT;
      "PREMIXING PROCESS" : Struct
         "PURIFIED WATER PROCESS SELECT" : Bool;
         "PURIFIED WATER PROCESS OF INITIAL DRAIN SELECT" : Bool;
         "PURIFIED WATER PROCESS OF LOAD CELL" : Bool;
         "PURIFIED WATER HEATING OR COOLING SELECT" : Bool;
         "PURIFIED WATER PROCESS OF JACKET DRAIN SELECT" : Bool;
         "PURIFIED WATER PROCESS OVER" : Bool;
         "MATERIAL ADDITION PROCESS SELECT" : Bool;
         "MATERIAL ADDITION MATERIAL ADDED TEXT" : Bool;
         "MATERIAL ADDITION DO YOU WANT TO ADD SORBITOL SELECT" : Bool;
         "MATERIAL ADDITION OF SORBITOL OVER" : Bool;
         "MATERIAL ADDITION DO YOU WANT TO ADD GLUCOSE SELECT" : Bool;
         "MATERIAL ADDITION OF GLUCOSE OVER" : Bool;
         "MATERIAL ADDITION PROCESS OVER" : Bool;
         "RECIRCULATION PROCESS SELECT" : Bool;
         "RECIRCULATION PROCESS RUNING" : Bool;
         "RECIRCULATION OVER" : Bool;
         "PREMIXING PROCESS OVER" : Bool;
      END_STRUCT;
      "PREMIXING PROCESS ALARM" : Struct
         "MFG PROCESS START" : Bool;
         "PURIFIED WATER PROCESS START" : Bool;
         "PURIFIED WATER PROCESS OF INITIAL DRAIN START" : Bool;
         "PURIFIED WATER PROCESS OF INITIAL DRAIN STOP" : Bool;
         "PURIFIED WATER PROCESS OF LOAD CELL START" : Bool;
         "PURIFIED WATER PROCESS OF LOAD CELL STOP" : Bool;
         "PURIFIED WATER OF HEATING START" : Bool;
         "PURIFIED WATER OF HEATING STOP" : Bool;
         "PURIFIED WATER OF COOLING START" : Bool;
         "PURIFIED WATER OF COOLING STOP" : Bool;
         "PURIFIED WATER PROCESS OF JACKET DRAIN START" : Bool;
         "PURIFIED WATER PROCESS OF JACKET DRAIN STOP" : Bool;
         "PURIFIED WATER PROCESS OVER" : Bool;
         "MATERIAL ADDITION PROCESS SELECT" : Bool;
         "MATERIAL ADDITION PROCESS START" : Bool;
         "MATERIAL ADDITION OF INITIAL DRAIN SELECT" : Bool;
         "MATERIAL ADDITION OF INITIAL DRAIN START" : Bool;
         "MATERIAL ADDITION OF INITIAL DRAIN STOP" : Bool;
         "MATERIAL ADDITION MATERIAL ADDED TEXT" : Bool;
         "MATERIAL ADDITION DO YOU WANT TO ADD SORBITOL SELECT" : Bool;
         "MATERIAL ADDITION OF SORBITOL START" : Bool;
         "MATERIAL ADDITION OF SORBITOL STIRRER START" : Bool;
         "MATERIAL ADDITION OF SORBITOL STIRRER STOP" : Bool;
         "MATERIAL ADDITION OF SORBITOL OVER" : Bool;
         "MATERIAL ADDITION DO YOU WANT TO ADD GLUCOSE SELECT" : Bool;
         "MATERIAL ADDITION OF GLUCOSE START" : Bool;
         "MATERIAL ADDITION OF GLUCOSE STIRRER START" : Bool;
         "MATERIAL ADDITION OF GLUCOSE STIRRER STOP" : Bool;
         "MATERIAL ADDITION OF GLUCOSE OVER" : Bool;
         "MATERIAL ADDITION PROCESS OF JACKET DRAIN SELECT" : Bool;
         "MATERIAL ADDITION PROCESS OF JACKET DRAIN STOP" : Bool;
         "MATERIAL ADDITION PROCESS OVER" : Bool;
         "RECIRCULATION PROCESS SELECT" : Bool;
         "RECIRCULATION PROCESS START" : Bool;
         "RECIRCULATION PROCESS OF INITIAL DRAIN SELECT" : Bool;
         "RECIRCULATION PROCESS OF INITIAL DRAIN START" : Bool;
         "RECIRCULATION PROCESS OF INITIAL DRAIN STOP" : Bool;
         "RECIRCULATION PROCESS RUNING" : Bool;
         "RECIRCULATION PROCESS OF JACKET DRAIN SELECT" : Bool;
         "RECIRCULATION PROCESS OF JACKET DRAIN STOP" : Bool;
         "RECIRCULATION OVER" : Bool;
         "MFG PROCESS OVER" : Bool;
      END_STRUCT;
      "PREMIXING TRANSFER START" : Struct
         "PREMIXING TO MFG WITH INLINE HOMO" : Bool;
         "PREMIXING TO MFG WITH INLINE FILTER PRES" : Bool;
         "PREMIXING TO STORAGE-4 WITH INLINE HOMO" : Bool;
         "PREMIXING TO STORAGE-4 WITH INLINE FILTER PRES" : Bool;
      END_STRUCT;
      "PREMIXING TRANSFER OVER" : Struct
         "PREMIXING TO MFG WITH INLINE HOMO" : Bool;
         "PREMIXING TO MFG WITH INLINE FILTER PRES" : Bool;
         "PREMIXING TO STORAGE-4 WITH INLINE HOMO" : Bool;
         "PREMIXING TO STORAGE-4 WITH INLINE FILTER PRES" : Bool;
      END_STRUCT;
      "PREMIXING MATERIAL SUCTION" : Struct
         "MATERIAL SUCTION START" : Bool;
         "MATERIAL SUCTION OVER" : Bool;
      END_STRUCT;
      "SUGAR PROCESS" : Struct
         "PURIFIED WATER PROCESS SELECT" : Bool;
         "PURIFIED WATER PROCESS OF INITIAL DRAIN SELECT" : Bool;
         "PURIFIED WATER PROCESS OF LOAD CELL" : Bool;
         "PURIFIED WATER HEATING OR COOLING SELECT" : Bool;
         "PURIFIED WATER PROCESS OF JACKET DRAIN SELECT" : Bool;
         "PURIFIED WATER PROCESS OVER" : Bool;
         "MATERIAL ADDITION PROCESS SELECT" : Bool;
         "MATERIAL ADDITION MATERIAL ADDED TEXT" : Bool;
         "MATERIAL ADDITION DO YOU WANT TO ADD SORBITOL SELECT" : Bool;
         "MATERIAL ADDITION OF SORBITOL OVER" : Bool;
         "MATERIAL ADDITION DO YOU WANT TO ADD GLUCOSE SELECT" : Bool;
         "MATERIAL ADDITION OF GLUCOSE OVER" : Bool;
         "MATERIAL ADDITION PROCESS OVER" : Bool;
         "RECIRCULATION PROCESS SELECT" : Bool;
         "RECIRCULATION PROCESS RUNING" : Bool;
         "RECIRCULATION OVER" : Bool;
         "MFG PROCESS OVER" : Bool;
      END_STRUCT;
      "SUGAR PROCESS ALARM" : Struct
         "MFG PROCESS START" : Bool;
         "PURIFIED WATER PROCESS START" : Bool;
         "PURIFIED WATER PROCESS OF INITIAL DRAIN START" : Bool;
         "PURIFIED WATER PROCESS OF INITIAL DRAIN STOP" : Bool;
         "PURIFIED WATER PROCESS OF LOAD CELL START" : Bool;
         "PURIFIED WATER PROCESS OF LOAD CELL STOP" : Bool;
         "PURIFIED WATER OF HEATING START" : Bool;
         "PURIFIED WATER OF HEATING STOP" : Bool;
         "PURIFIED WATER OF COOLING START" : Bool;
         "PURIFIED WATER OF COOLING STOP" : Bool;
         "PURIFIED WATER PROCESS OF JACKET DRAIN START" : Bool;
         "PURIFIED WATER PROCESS OF JACKET DRAIN STOP" : Bool;
         "PURIFIED WATER PROCESS OVER" : Bool;
         "MATERIAL ADDITION PROCESS SELECT" : Bool;
         "MATERIAL ADDITION PROCESS START" : Bool;
         "MATERIAL ADDITION OF INITIAL DRAIN SELECT" : Bool;
         "MATERIAL ADDITION OF INITIAL DRAIN START" : Bool;
         "MATERIAL ADDITION OF INITIAL DRAIN STOP" : Bool;
         "MATERIAL ADDITION MATERIAL ADDED TEXT" : Bool;
         "MATERIAL ADDITION DO YOU WANT TO ADD SORBITOL SELECT" : Bool;
         "MATERIAL ADDITION OF SORBITOL START" : Bool;
         "MATERIAL ADDITION OF SORBITOL STIRRER START" : Bool;
         "MATERIAL ADDITION OF SORBITOL STIRRER STOP" : Bool;
         "MATERIAL ADDITION OF SORBITOL OVER" : Bool;
         "MATERIAL ADDITION DO YOU WANT TO ADD GLUCOSE SELECT" : Bool;
         "MATERIAL ADDITION OF GLUCOSE START" : Bool;
         "MATERIAL ADDITION OF GLUCOSE STIRRER START" : Bool;
         "MATERIAL ADDITION OF GLUCOSE STIRRER STOP" : Bool;
         "MATERIAL ADDITION OF GLUCOSE OVER" : Bool;
         "MATERIAL ADDITION PROCESS OF JACKET DRAIN SELECT" : Bool;
         "MATERIAL ADDITION PROCESS OF JACKET DRAIN STOP" : Bool;
         "MATERIAL ADDITION PROCESS OVER" : Bool;
         "RECIRCULATION PROCESS SELECT" : Bool;
         "RECIRCULATION PROCESS START" : Bool;
         "RECIRCULATION PROCESS OF INITIAL DRAIN SELECT" : Bool;
         "RECIRCULATION PROCESS OF INITIAL DRAIN START" : Bool;
         "RECIRCULATION PROCESS OF INITIAL DRAIN STOP" : Bool;
         "RECIRCULATION PROCESS RUNING" : Bool;
         "RECIRCULATION PROCESS OF JACKET DRAIN SELECT" : Bool;
         "RECIRCULATION PROCESS OF JACKET DRAIN STOP" : Bool;
         "RECIRCULATION OVER" : Bool;
         "MFG PROCESS OVER" : Bool;
      END_STRUCT;
      "SUGAR TRANSFER START" : Struct
         "PREMIXING TO MFG WITH INLINE HOMO" : Bool;
         "PREMIXING TO MFG WITH INLINE FILTER PRES" : Bool;
         "PREMIXING TO STORAGE-4 WITH INLINE HOMO" : Bool;
         "PREMIXING TO STORAGE-4 WITH INLINE FILTER PRES" : Bool;
      END_STRUCT;
      "SUGAR TRANSFER OVER" : Struct
         "PREMIXING TO MFG WITH INLINE HOMO" : Bool;
         "PREMIXING TO MFG WITH INLINE FILTER PRES" : Bool;
         "PREMIXING TO STORAGE-4 WITH INLINE HOMO" : Bool;
         "PREMIXING TO STORAGE-4 WITH INLINE FILTER PRES" : Bool;
      END_STRUCT;
      "SUGAR MATERIAL SUCTION" : Struct
         "MATERIAL SUCTION START" : Bool;
         "MATERIAL SUCTION OVER" : Bool;
      END_STRUCT;
   END_VAR
BEGIN
END_DATA_BLOCK

DATA_BLOCK "AUTO P_TRIG"   // DB71
{ S7_Optimized_Access := 'TRUE' }
// stored: MemoryReserve 100
   VAR
      "1" : Bool;
      "2" : Bool;
      "3" : Bool;
      "4" : Bool;
      "5" : Bool;
      "6" : Bool;
      "7" : Bool;
      "8" : Bool;
      "9" : Bool;
      "10" : Bool;
      "11" : Bool;
      "12" : Bool;
      "13" : Bool;
      "14" : Bool;
      "15" : Bool;
      "16" : Bool;
      "17" : Bool;
      "18" : Bool;
      "19" : Bool;
      "20" : Bool;
      "21" : Bool;
      "22" : Bool;
      "23" : Bool;
      "24" : Bool;
      "25" : Bool;
      "26" : Bool;
      "27" : Bool;
      "28" : Bool;
      "29" : Bool;
      "30" : Bool;
   END_VAR
BEGIN
END_DATA_BLOCK

DATA_BLOCK "P_TRIG"   // DB10
{ S7_Optimized_Access := 'TRUE' }
// stored: MemoryReserve 100
   VAR
      "1" : Bool;
      "2" : Bool;
      "3" : Bool;
      "4" : Bool;
      "5" : Bool;
      "6" : Bool;
      "7" : Bool;
      "8" : Bool;
      "9" : Bool;
      "10" : Bool;
      "11" : Bool;
      "12" : Bool;
      "13" : Bool;
      "14" : Bool;
      "15" : Bool;
      "16" : Bool;
      "17" : Bool;
      "18" : Bool;
      "19" : Bool;
      "20" : Bool;
      "21" : Bool;
      "22" : Bool;
      "23" : Bool;
      "24" : Bool;
      "25" : Bool;
      "26" : Bool;
      "27" : Bool;
      "28" : Bool;
      "29" : Bool;
      "30" : Bool;
      "31" : Bool;
      "32" : Bool;
      "33" : Bool;
      "34" : Bool;
      "35" : Bool;
      "36" : Bool;
      "37" : Bool;
      "38" : Bool;
      "39" : Bool;
      "40" : Bool;
      "41" : Bool;
      "42" : Bool;
      "43" : Bool;
      "44" : Bool;
      "45" : Bool;
      "46" : Bool;
      "47" : Bool;
      "48" : Bool;
      "49" : Bool;
      "50" : Bool;
      "51" : Bool;
      "52" : Bool;
      "53" : Bool;
      "54" : Bool;
      "55" : Bool;
      "56" : Bool;
      "57" : Bool;
      "58" : Bool;
      "59" : Bool;
      "60" : Bool;
      "61" : Bool;
      "62" : Bool;
   END_VAR
BEGIN
END_DATA_BLOCK

DATA_BLOCK "CONTINUE DB"   // DB11
{ S7_Optimized_Access := 'TRUE' }
// stored: MemoryReserve 100
   VAR RETAIN
      "SYRUP MFG PROCESS ERROR" : Int;
      "PREMIXING PROCESS ERROR" : Int;
      "SUGAR PROCESS ERROR" : Int;
      "MFG PROCESS CONTINUE" : Bool;
      "MFG PROCESS RESET" : Bool;
      "PREMIX PROCESS CONTINUE" : Bool;
      "PREMIX PROCESS RESET" : Bool;
      "SUGAR PROCESS CONTINUE" : Bool;
      "SUGAR PREMIX PROCESS RESET" : Bool;
   END_VAR
BEGIN
END_DATA_BLOCK

DATA_BLOCK "HYST AND TEMP CUTOFF  DB"   // DB13
{ S7_Optimized_Access := 'TRUE' }
// stored: MemoryReserve 100
   VAR RETAIN
      "MAN SET" : Struct
         "SYRUP MFG_TEMP" : Real;
         "SYRUP MFG_COOLING" : Real;
         "SYRUP MFG_VACCUM" : Real;
         "SYRUP MFG_LOAD CELL" : Real;
         "MFG MOVE PV LOAD CELL" : Real;
         PREMIXING_TEMP : Real;
         PREMIXING_COOLING : Real;
         PREMIXING_VACCUM : Real;
         "PREMIXING_LOAD CELL" : Real;
         "PREMIXING MOVE PV LOAD CELL" : Real;
         SUGAR_TEMP : Real;
         SUGAR_VACCUM : Real;
         "SUGAR_LOAD CELL" : Real;
         "SUGAR MOVE PV LOAD CELL" : Real;
      END_STRUCT;
      "MAIN SET PARA" : Struct
         "SYRUP MFG_TEMP" : Real;
         "SYRUP MFG_COOLING" : Real;
         "SYRUP MFG_VACCUM" : Real;
         "SYRUP MFG_LOAD CELL" : Real;
         "AUTO MFG_LOAD CELL" : Real;
         PREMIXING_TEMP : Real;
         PREMIXING_COOING : Real;
         PREMIXING_VACCUM : Real;
         "PREMIXING_LOAD CELL" : Real;
         "AUTO PREMIXING_LOAD CELL" : Real;
         SUGAR_TEMP : Real;
         SUGAR_VACCUM : Real;
         "SUGAR_LOAD CELL" : Real;
         "AUTO SUGAR_LOAD CELL" : Real;
      END_STRUCT;
      "HYSTERISIS SUB" : Struct
         "SYRUP MFG_TEMP" : Real;
         "SYRUP MFG_COOLING" : Real;
         "SYRUP MFG_VACCUM" : Real;
         "SYRUP MFG_LOAD CELL" : Real;
         PREMIXING_TEMP : Real;
         PREMIXING_COOLING : Real;
         PREMIXING_VACCUM : Real;
         "PREMIXING_LOAD CELL" : Real;
         SUGAR_TEMP : Real;
         SUGAR_VACCUM : Real;
         "SUGAR_LOAD CELL" : Real;
      END_STRUCT;
      "HYSTERISIS NEW_VALUE" : Struct
         "SYRUP MFG_TEMP" : Real;
         "SYRUP MFG_COOLING" : Real;
         "SYRUP MFG_VACCUM" : Real;
         "SYRUP MFG_LOAD CELL" : Real;
         "AUTO MFG_LOAD CELL" : Real;
         PREMIXING_TEMP : Real;
         PREMIXING_COOLING : Real;
         PREMIXING_VACCUM : Real;
         "PREMIXING_LOAD CELL" : Real;
         "AUTO PREMIXING_LOAD CELL" : Real;
         SUGAR_TEMP : Real;
         SUGAR_VACCUM : Real;
         "SUGAR_LOAD CELL" : Real;
         "AUTO SUGAR_LOAD CELL" : Real;
      END_STRUCT;
      "MFG CALCULATE PV" : Real;
      "PREMIXING CALCULATE PV" : Real;
      "SUGAR CALCULATE PV" : Real;
      "AUTO SET" : Struct
         MFG_TEMP : Real;
         MFG_COOLING : Real;
         MFG_VACCUM : Real;
         "MFG_LOAD CELL" : Real;
         "MFG LOAD CELL FOR TRANSFER" : Real;
         PREMIXING_TEMP : Real;
         PREMIXING_COOLING : Real;
         PREMIXING_VACCUM : Real;
         "PREMIXING_LOAD CELL" : Real;
         "PREMIXING LOAD CELL FOR TRANSFER" : Real;
         SUGAR_TEMP : Real;
         SUGAR_VACCUM : Real;
         "SUGAR_LOAD CELL" : Real;
         "SUGAR LOAD CELL FOR TRANSFER" : Real;
      END_STRUCT;
      "AUTO MAIN SET PARAMETER" : Struct
         "MFG LOAD CELL" : Real;
         "PREMIXING LOAD CELL" : Real;
         "SUGAR LOAD CELL" : Real;
      END_STRUCT;
      "AUTO NEW VALUE" : Struct
         "MFG LOAD CELL" : Real;
         "PREMIXING LOAD CELL" : Real;
         "SUGAR LOAD CELL" : Real;
      END_STRUCT;
      "AUTO MOVE PV" : Struct
         "MFG_LOAD CELL" : Real;
         "PREMIXING_LOAD CELL" : Real;
         "SUGAR_LOAD CELL" : Real;
      END_STRUCT;
   END_VAR
   VAR
      "MIAN MFG TEMP MIN" : Real;
      "MIAN MFG TEMP MAX" : Real;
      "MIAN PREMIXING TEMP MIN" : Real;
      "MIAN PREMIXING TEMP MAX" : Real;
   END_VAR
BEGIN
END_DATA_BLOCK

DATA_BLOCK "LEVEL BUFF"   // DB14
{ S7_Optimized_Access := 'TRUE' }
// stored: MemoryReserve 100
   VAR RETAIN
      "SYRUP MFG_TEMP" : Int;
      "SYRUP MFG_COOLING" : Int;
      "SYRUP MFG_VACCUM" : Int;
      "SYRUP MFG_LOAD CELL" : Int;
      PREMIXING_TEMP : Int;
      PREMIXING_COOLING : Int;
      PREMIXING_VACCUM : Int;
      "PREMIXING_LOAD CELL" : Int;
      SUGAR_TEMP : Int;
      SUGAR_VACCUM : Int;
      "SUGAR_LOAD CELL" : Int;
   END_VAR
   VAR
      AUTO : Struct
         "MFG LOAD CELL" : Int;
         "MFG TEMP MIN_MAX BUFF" : Int;
         "MFG VACUUM MIN_MAX BUFF" : Int;
         "PREMIXING LOAD CELL" : Int;
         "PREMIXING TEMP MIN_MAX BUFF" : Int;
         "PREMIXING VACUUM MIN_MAX BUFF" : Int;
         "SUGAR LOAD CELL" : Int;
         "SUGAR TEMP MIN_MAX BUFF" : Int;
         "SUGAR VACUUM MIN_MAX BUFF" : Int;
      END_STRUCT;
   END_VAR
BEGIN
END_DATA_BLOCK

DATA_BLOCK "SET PARAMETER DB"   // DB44
{ S7_Optimized_Access := 'TRUE' }
// stored: MemoryReserve 100
   VAR RETAIN
      "MANUAL VFD SET PARAMETER" : Struct
         "MFG VESSEL STIRROR RUN" : Real;
         "PREMIXING  VESSEL STIRROR RUN" : Real;
         "SUGAR VESSEL STIRROR RUN" : Real;
      END_STRUCT;
   END_VAR
   VAR
      "AUTO VFD SET PARAMETER" : Struct
         "MFG VESSEL STIRROR RUN" : Real;
         "PREMIXING  VESSEL STIRROR RUN" : Real;
         "SUGAR VESSEL STIRROR RUN" : Real;
      END_STRUCT;
   END_VAR
BEGIN
END_DATA_BLOCK

ORGANIZATION_BLOCK "Main"   // OB1, LAD, ProgramCycle
TITLE = "Main Program Sweep (Cycle)"
{ S7_Optimized_Access := 'TRUE' }
// stored: SetENOAutomatically false
   VAR_INPUT
      Initial_Call : Bool;   // Initial call of this OB
      Remanence : Bool;   // =True, if remanent data are available
   END_VAR
   VAR_TEMP   // added for the SCL form of the ladder/FBD networks
      _w1 : Bool;
      _w2 : Bool;
      _w3 : Bool;
      _w4 : Bool;
      _w5 : Bool;
      _w6 : Bool;
      _w7 : Bool;
      _w8 : Bool;
      _w9 : Bool;
      _w10 : Bool;
   END_VAR
BEGIN

REGION Network 1: #SHIV
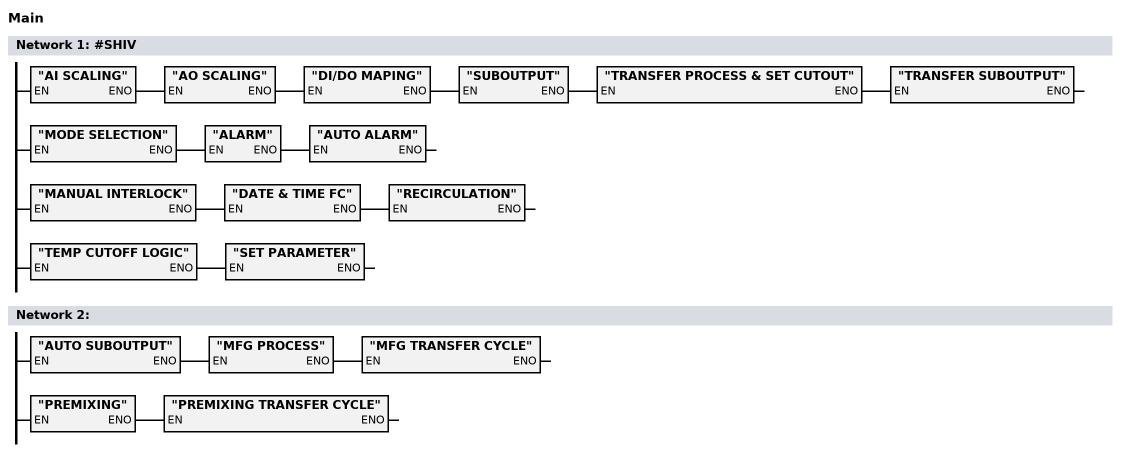
   RUNG wire#powerrail
      "AI SCALING"()
      "AO SCALING"()
      "DI/DO MAPING"()
      "SUBOUTPUT"()
      "TRANSFER PROCESS & SET CUTOUT"()
      "TRANSFER SUBOUTPUT"()
   END_RUNG
   RUNG wire#powerrail
      "MODE SELECTION"()
      "ALARM"()
      "AUTO ALARM"()
   END_RUNG
   RUNG wire#powerrail
      "MANUAL INTERLOCK"()
      "DATE & TIME FC"()
      "RECIRCULATION"()
   END_RUNG
   RUNG wire#powerrail
      "TEMP CUTOFF LOGIC"()
      "SET PARAMETER"()
   END_RUNG
   // the same network as SCL:
   "AI SCALING"(ENO => #_w1);
   "AO SCALING"(EN := #_w1, ENO => #_w2);
   "DI/DO MAPING"(EN := #_w2, ENO => #_w3);
   "SUBOUTPUT"(EN := #_w3, ENO => #_w4);
   "TRANSFER PROCESS & SET CUTOUT"(EN := #_w4, ENO => #_w5);
   IF #_w5 THEN "TRANSFER SUBOUTPUT"(); END_IF;
   "MODE SELECTION"(ENO => #_w6);
   "ALARM"(EN := #_w6, ENO => #_w7);
   IF #_w7 THEN "AUTO ALARM"(); END_IF;
   "MANUAL INTERLOCK"(ENO => #_w8);
   "DATE & TIME FC"(EN := #_w8, ENO => #_w9);
   IF #_w9 THEN "RECIRCULATION"(); END_IF;
   "TEMP CUTOFF LOGIC"(ENO => #_w10);
   IF #_w10 THEN "SET PARAMETER"(); END_IF;
END_REGION

REGION Network 2
   RUNG wire#powerrail
      "AUTO SUBOUTPUT"()
      "MFG PROCESS"()
      "MFG TRANSFER CYCLE"()
   END_RUNG
   RUNG wire#powerrail
      "PREMIXING"()
      "PREMIXING TRANSFER CYCLE"()
   END_RUNG
   // the same network as SCL:
   "AUTO SUBOUTPUT"(ENO => #_w1);
   "MFG PROCESS"(EN := #_w1, ENO => #_w2);
   IF #_w2 THEN "MFG TRANSFER CYCLE"(); END_IF;
   "PREMIXING"(ENO => #_w3);
   IF #_w3 THEN "PREMIXING TRANSFER CYCLE"(); END_IF;
END_REGION
END_ORGANIZATION_BLOCK

FUNCTION "AO SCALING" : Void
{ S7_Optimized_Access := 'TRUE' }
VERSION : 0.1

BEGIN
	REGION SYRUP MFG VESSEL SPEED
	    IF "DO MAPING"."SYRUP MFG VESSEL BOTTOM STERROR RUN" = FALSE THEN
	        "SYRUP MFG VESSEL SPEED" := 0;
	        "AO SCALING DB".PV."SYRUP MFG VESSEL SPEED" := 0.0;
	    ELSE
	        "@SCALING AO"("ANALOG OUTPUT" := "AO SCALING DB".SET."SYRUP MFG VESSEL SPEED",
	                      "SCALING MIN" := "AO SCALING DB".MIN."SYRUP MFG VESSEL SPEED",
	                      "SCALING MAX" := "AO SCALING DB".MAX."SYRUP MFG VESSEL SPEED",
	                      "RAW MIN" := 0,
	                      "RAW MAX" := 27648,
	                      "PV VALUE" => "SYRUP MFG VESSEL SPEED");
	        "@SCALING AI"("ANALOG INPUT" := "SYRUP MFG VESSEL SPEED",
	                      "RAW MIN" := 0,
	                      "RAW MAX" := 27648,
	                      "SCALE MIN" := "AO SCALING DB".MIN."SYRUP MFG VESSEL SPEED",
	                      "SCALE MAX" := "AO SCALING DB".MAX."SYRUP MFG VESSEL SPEED",
	                      "PV VALUE" => "AO SCALING DB".PV."SYRUP MFG VESSEL SPEED");
	        ;
	    END_IF;
	
	    CASE "MODE SELECTION DB"."MODE BUFF" OF
	        1:  "AO SCALING DB".SET."SYRUP MFG VESSEL SPEED" :=
	            "SET PARAMETER DB"."AUTO VFD SET PARAMETER"."MFG VESSEL STIRROR RUN"
	            ;
	        2:
	            "AO SCALING DB".SET."SYRUP MFG VESSEL SPEED" :=
	            "SET PARAMETER DB"."MANUAL VFD SET PARAMETER"."MFG VESSEL STIRROR RUN";
	            ;
	        ELSE
	            "AO SCALING DB".SET."SYRUP MFG VESSEL SPEED" := 0.0;
	            ;
	    END_CASE;
	    
	END_REGION
	
	REGION PREMIXING VESSEL SPEED
	    IF "DO MAPING"."PREMIXING VESSEL BOTTOM STERROR RUN" = FALSE THEN
	        "PREMIXING VESSEL SPEED" := 0;
	        "AO SCALING DB".PV."PREMIXING VESSEL SPEED" := 0.0;
	    ELSE
	        "@SCALING AO"("ANALOG OUTPUT" := "AO SCALING DB".SET."PREMIXING VESSEL SPEED",
	                      "SCALING MIN" := "AO SCALING DB".MIN."PREMIXING VESSEL SPEED",
	                      "SCALING MAX" := "AO SCALING DB".MAX."PREMIXING VESSEL SPEED",
	                      "RAW MIN" := 0,
	                      "RAW MAX" := 27648,
	                      "PV VALUE" => "PREMIXING VESSEL SPEED");
	        "@SCALING AI"("ANALOG INPUT" := "PREMIXING VESSEL SPEED",
	                      "RAW MIN" := 0,
	                      "RAW MAX" := 27648,
	                      "SCALE MIN" := "AO SCALING DB".MIN."PREMIXING VESSEL SPEED",
	                      "SCALE MAX" := "AO SCALING DB".MAX."PREMIXING VESSEL SPEED",
	                      "PV VALUE" => "AO SCALING DB".PV."PREMIXING VESSEL SPEED");
	        ;
	    END_IF;
	    CASE "MODE SELECTION DB"."MODE BUFF" OF
	        1:
	            "AO SCALING DB".SET."PREMIXING VESSEL SPEED" :=
	            "SET PARAMETER DB"."AUTO VFD SET PARAMETER"."PREMIXING  VESSEL STIRROR RUN"
	            ;
	        2:
	            "AO SCALING DB".SET."PREMIXING VESSEL SPEED" :=
	            "SET PARAMETER DB"."MANUAL VFD SET PARAMETER"."PREMIXING  VESSEL STIRROR RUN";
	            ;
	        ELSE
	            "AO SCALING DB".SET."PREMIXING VESSEL SPEED" := 0.0;
	            ;
	    END_CASE;
	END_REGION
	
	REGION SUGAR VESSEL SPEED
	    IF "DO MAPING"."SUGAR VESSEL BOTTOM STERROR RUN" = FALSE THEN
	        "SUGAR VESSEL SPEED" := 0;
	        "AO SCALING DB".PV."SUGAR VESSEL SPEED" := 0.0;
	    ELSE
	        "@SCALING AO"("ANALOG OUTPUT" := "AO SCALING DB".SET."SUGAR VESSEL SPEED",
	                      "SCALING MIN" := "AO SCALING DB".MIN."SUGAR VESSEL SPEED",
	                      "SCALING MAX" := "AO SCALING DB".MAX."SUGAR VESSEL SPEED",
	                      "RAW MIN" := 0,
	                      "RAW MAX" := 27648,
	                      "PV VALUE" => "SUGAR VESSEL SPEED");
	        "@SCALING AI"("ANALOG INPUT" := "SUGAR VESSEL SPEED",
	                      "RAW MIN" := 0,
	                      "RAW MAX" := 27648,
	                      "SCALE MIN" := "AO SCALING DB".MIN."SUGAR VESSEL SPEED",
	                      "SCALE MAX" := "AO SCALING DB".MAX."SUGAR VESSEL SPEED",
	                      "PV VALUE" => "AO SCALING DB".PV."SUGAR VESSEL SPEED");
	        ;
	    END_IF;
	    CASE "MODE SELECTION DB"."MODE BUFF" OF
	        1:
	            "AO SCALING DB".SET."SUGAR VESSEL SPEED" :=
	            "SET PARAMETER DB"."AUTO VFD SET PARAMETER"."SUGAR VESSEL STIRROR RUN"
	            ;
	        2:
	            "AO SCALING DB".SET."SUGAR VESSEL SPEED" :=
	            "SET PARAMETER DB"."MANUAL VFD SET PARAMETER"."SUGAR VESSEL STIRROR RUN";
	            ;
	        ELSE
	            "AO SCALING DB".SET."SUGAR VESSEL SPEED" := 0.0;
	            ;
	    END_CASE;
	END_REGION
	
	
	
	
	
	
	
	
	
	
	
	
	
	
	
	
	
	
	
	
	
	
END_FUNCTION

FUNCTION "TRANSFER PROCESS & SET CUTOUT" : Void   // FC12, LAD
{ S7_Optimized_Access := 'TRUE' }
// stored: SetENOAutomatically false
   VAR_TEMP   // added for the SCL form of the ladder/FBD networks
      _w1 : Bool;
      _w2 : Bool;
   END_VAR
BEGIN

REGION Network 1 (SCL): MFG VESSEL STIRRER RUN
   REGION MFG VESSEL STIRRER RUN

       IF ("MANUAL TIME BASE DB"."MFG VESSEL STIRRER RUN".SV = 0) OR
           ("MANUAL BIT"."SYRUP MFG VESSEL BOTTOM STERROR RUN" = 1 AND "TIMER_MIN_DB".DONE)
       THEN
           "MANUAL BIT"."SYRUP MFG VESSEL BOTTOM STERROR RUN" := FALSE;
       ELSE
           "TIMER_MIN_DB"("SET TIME" := "MANUAL TIME BASE DB"."MFG VESSEL STIRRER RUN".SV,
                          RESET := "TIMER_MIN_DB".RESET,
                          INPUT := "MANUAL BIT"."SYRUP MFG VESSEL BOTTOM STERROR RUN",
                          "PRESENT VALUE OF TIME" => "MANUAL TIME BASE DB"."MFG VESSEL STIRRER RUN".PV);
       END_IF;
       IF "MODE SELECTION DB"."MODE BUFF" <> 2 OR
           "MANUAL TIME BASE DB"."MFG VESSEL STIRRER RUN"."RESET TIME" = TRUE THEN
           "TIMER_MIN_DB".RESET := TRUE;
       ELSE
           "TIMER_MIN_DB".RESET := FALSE;
       END_IF;
   END_REGION
END_REGION

REGION Network 2 (SCL): PREMIXING VESSEL STIRRER RUN
   REGION PREMIXING  VESSEL STIRRER RUN

       IF ("MANUAL TIME BASE DB"."PREMIXING  VESSEL STIRRER RUN".SV = 0) OR
           ("MANUAL BIT"."PREMIXING VESSEL BOTTOM STERROR RUN" = 1 AND "TIMER_MIN_DB_1".DONE)
       THEN
           "MANUAL BIT"."PREMIXING VESSEL BOTTOM STERROR RUN" := FALSE;
       ELSE
           "TIMER_MIN_DB_1"("SET TIME" := "MANUAL TIME BASE DB"."PREMIXING  VESSEL STIRRER RUN".SV,
                            RESET := "TIMER_MIN_DB_1".RESET,
                            INPUT := "MANUAL BIT"."PREMIXING VESSEL BOTTOM STERROR RUN",
                            "PRESENT VALUE OF TIME" => "MANUAL TIME BASE DB"."PREMIXING  VESSEL STIRRER RUN".PV);
       END_IF;
       IF "MODE SELECTION DB"."MODE BUFF" <> 2 OR
           "MANUAL TIME BASE DB"."PREMIXING  VESSEL STIRRER RUN"."RESET TIME" = TRUE THEN
           "TIMER_MIN_DB_1".RESET := TRUE;
       ELSE
           "TIMER_MIN_DB_1".RESET := FALSE;
       END_IF;
   END_REGION
END_REGION

REGION Network 3 (SCL): SUGAR VESSEL STIRRER RUN
   REGION SUGAR VESSEL STIRRER RUN

       IF ("MANUAL TIME BASE DB"."SUGAR VESSEL STIRRER RUN".SV = 0) OR
           ("MANUAL BIT"."SUGAR VESSEL BOTTOM STERROR RUN" = 1 AND "TIMER_MIN_DB_2".DONE)
       THEN
           "MANUAL BIT"."SUGAR VESSEL BOTTOM STERROR RUN" := FALSE;
       ELSE
           "TIMER_MIN_DB_2"("SET TIME" := "MANUAL TIME BASE DB"."SUGAR VESSEL STIRRER RUN".SV,
                            RESET := "TIMER_MIN_DB_2".RESET,
                            INPUT := "MANUAL BIT"."SUGAR VESSEL BOTTOM STERROR RUN",
                            "PRESENT VALUE OF TIME" => "MANUAL TIME BASE DB"."SUGAR VESSEL STIRRER RUN".PV);
       END_IF;
       IF "MODE SELECTION DB"."MODE BUFF" <> 2 OR
           "MANUAL TIME BASE DB"."SUGAR VESSEL STIRRER RUN"."RESET TIME" = TRUE THEN
           "TIMER_MIN_DB_2".RESET := TRUE;
       ELSE
           "TIMER_MIN_DB_2".RESET := FALSE;
       END_IF;
   END_REGION
END_REGION

REGION Network 5: SYRUP MFG_TEMP_CUTOUT
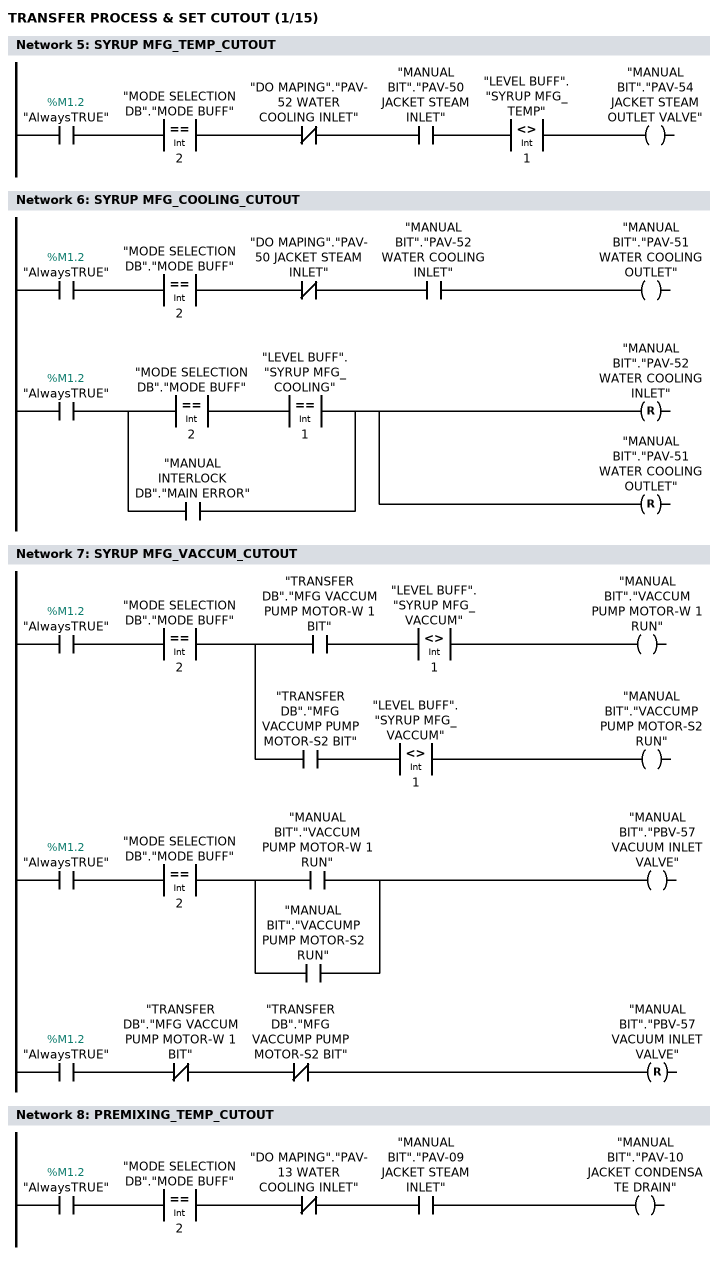
   RUNG wire#powerrail
      Contact( "AlwaysTRUE" )
      { S7_Templates := "SrcType := Int" } EQ_Contact(in1 := "MODE SELECTION DB"."MODE BUFF", in2 := 2)
      I_Contact( "DO MAPING"."PAV-52 WATER COOLING INLET" )
      Contact( "MANUAL BIT"."PAV-50 JACKET STEAM INLET" )
      { S7_Templates := "SrcType := Int" } NE_Contact(in1 := "LEVEL BUFF"."SYRUP MFG_TEMP", in2 := 1)
      Coil( "MANUAL BIT"."PAV-54 JACKET STEAM OUTLET VALVE" )
   END_RUNG
   // the same network as SCL:
   "MANUAL BIT"."PAV-54 JACKET STEAM OUTLET VALVE" := "AlwaysTRUE" AND ("MODE SELECTION DB"."MODE BUFF" = 2) AND NOT "DO MAPING"."PAV-52 WATER COOLING INLET" AND "MANUAL BIT"."PAV-50 JACKET STEAM INLET" AND ("LEVEL BUFF"."SYRUP MFG_TEMP" <> 1);
END_REGION

REGION Network 6: SYRUP MFG_COOLING_CUTOUT
   RUNG wire#powerrail
      Contact( "AlwaysTRUE" )
      { S7_Templates := "SrcType := Int" } EQ_Contact(in1 := "MODE SELECTION DB"."MODE BUFF", in2 := 2)
      I_Contact( "DO MAPING"."PAV-50 JACKET STEAM INLET" )
      Contact( "MANUAL BIT"."PAV-52 WATER COOLING INLET" )
      Coil( "MANUAL BIT"."PAV-51 WATER COOLING OUTLET" )
   END_RUNG
   RUNG wire#powerrail
      Contact( "AlwaysTRUE" )
      wire#w1
      { S7_Templates := "SrcType := Int" } EQ_Contact(in1 := "MODE SELECTION DB"."MODE BUFF", in2 := 2)
      { S7_Templates := "SrcType := Int" } EQ_Contact(in1 := "LEVEL BUFF"."SYRUP MFG_COOLING", in2 := 1)
      wire#w2
      R_Coil( "MANUAL BIT"."PAV-52 WATER COOLING INLET" )
   END_RUNG
   RUNG wire#w1
      Contact( "MANUAL INTERLOCK DB"."MAIN ERROR" )
   END_RUNG wire#w2
   RUNG wire#w2
      R_Coil( "MANUAL BIT"."PAV-51 WATER COOLING OUTLET" )
   END_RUNG
   // the same network as SCL:
   "MANUAL BIT"."PAV-51 WATER COOLING OUTLET" := "AlwaysTRUE" AND ("MODE SELECTION DB"."MODE BUFF" = 2) AND NOT "DO MAPING"."PAV-50 JACKET STEAM INLET" AND "MANUAL BIT"."PAV-52 WATER COOLING INLET";
   IF "AlwaysTRUE" AND ((("MODE SELECTION DB"."MODE BUFF" = 2) AND ("LEVEL BUFF"."SYRUP MFG_COOLING" = 1)) OR "MANUAL INTERLOCK DB"."MAIN ERROR") THEN
       "MANUAL BIT"."PAV-52 WATER COOLING INLET" := FALSE;
       "MANUAL BIT"."PAV-51 WATER COOLING OUTLET" := FALSE;
   END_IF;
END_REGION

REGION Network 7: SYRUP MFG_VACCUM_CUTOUT
   RUNG wire#powerrail
      Contact( "AlwaysTRUE" )
      { S7_Templates := "SrcType := Int" } EQ_Contact(in1 := "MODE SELECTION DB"."MODE BUFF", in2 := 2)
      wire#w1
      Contact( "TRANSFER DB"."MFG VACCUM PUMP MOTOR-W 1 BIT" )
      { S7_Templates := "SrcType := Int" } NE_Contact(in1 := "LEVEL BUFF"."SYRUP MFG_VACCUM", in2 := 1)
      Coil( "MANUAL BIT"."VACCUM PUMP MOTOR-W 1 RUN" )
   END_RUNG
   RUNG wire#w1
      Contact( "TRANSFER DB"."MFG VACCUMP PUMP MOTOR-S2 BIT" )
      { S7_Templates := "SrcType := Int" } NE_Contact(in1 := "LEVEL BUFF"."SYRUP MFG_VACCUM", in2 := 1)
      Coil( "MANUAL BIT"."VACCUMP PUMP MOTOR-S2 RUN" )
   END_RUNG
   RUNG wire#powerrail
      Contact( "AlwaysTRUE" )
      { S7_Templates := "SrcType := Int" } EQ_Contact(in1 := "MODE SELECTION DB"."MODE BUFF", in2 := 2)
      wire#w2
      Contact( "MANUAL BIT"."VACCUM PUMP MOTOR-W 1 RUN" )
      wire#w3
      Coil( "MANUAL BIT"."PBV-57 VACUUM INLET VALVE" )
   END_RUNG
   RUNG wire#w2
      Contact( "MANUAL BIT"."VACCUMP PUMP MOTOR-S2 RUN" )
   END_RUNG wire#w3
   RUNG wire#powerrail
      Contact( "AlwaysTRUE" )
      I_Contact( "TRANSFER DB"."MFG VACCUM PUMP MOTOR-W 1 BIT" )
      I_Contact( "TRANSFER DB"."MFG VACCUMP PUMP MOTOR-S2 BIT" )
      R_Coil( "MANUAL BIT"."PBV-57 VACUUM INLET VALVE" )
   END_RUNG
   // the same network as SCL:
   #_w1 := "AlwaysTRUE" AND ("MODE SELECTION DB"."MODE BUFF" = 2);
   "MANUAL BIT"."VACCUM PUMP MOTOR-W 1 RUN" := #_w1 AND "TRANSFER DB"."MFG VACCUM PUMP MOTOR-W 1 BIT" AND ("LEVEL BUFF"."SYRUP MFG_VACCUM" <> 1);
   "MANUAL BIT"."VACCUMP PUMP MOTOR-S2 RUN" := #_w1 AND "TRANSFER DB"."MFG VACCUMP PUMP MOTOR-S2 BIT" AND ("LEVEL BUFF"."SYRUP MFG_VACCUM" <> 1);
   "MANUAL BIT"."PBV-57 VACUUM INLET VALVE" := "AlwaysTRUE" AND ("MODE SELECTION DB"."MODE BUFF" = 2) AND ("MANUAL BIT"."VACCUM PUMP MOTOR-W 1 RUN" OR "MANUAL BIT"."VACCUMP PUMP MOTOR-S2 RUN");
   IF "AlwaysTRUE" AND NOT "TRANSFER DB"."MFG VACCUM PUMP MOTOR-W 1 BIT" AND NOT "TRANSFER DB"."MFG VACCUMP PUMP MOTOR-S2 BIT" THEN
       "MANUAL BIT"."PBV-57 VACUUM INLET VALVE" := FALSE;
   END_IF;
END_REGION

REGION Network 8: PREMIXING_TEMP_CUTOUT
   RUNG wire#powerrail
      Contact( "AlwaysTRUE" )
      { S7_Templates := "SrcType := Int" } EQ_Contact(in1 := "MODE SELECTION DB"."MODE BUFF", in2 := 2)
      I_Contact( "DO MAPING"."PAV-13 WATER COOLING INLET" )
      Contact( "MANUAL BIT"."PAV-09 JACKET STEAM INLET" )
      Coil( "MANUAL BIT"."PAV-10 JACKET CONDENSATE DRAIN" )
   END_RUNG
   // the same network as SCL:
   "MANUAL BIT"."PAV-10 JACKET CONDENSATE DRAIN" := "AlwaysTRUE" AND ("MODE SELECTION DB"."MODE BUFF" = 2) AND NOT "DO MAPING"."PAV-13 WATER COOLING INLET" AND "MANUAL BIT"."PAV-09 JACKET STEAM INLET";
END_REGION

REGION Network 9: PREMIXING_COOLING_CUTOUT
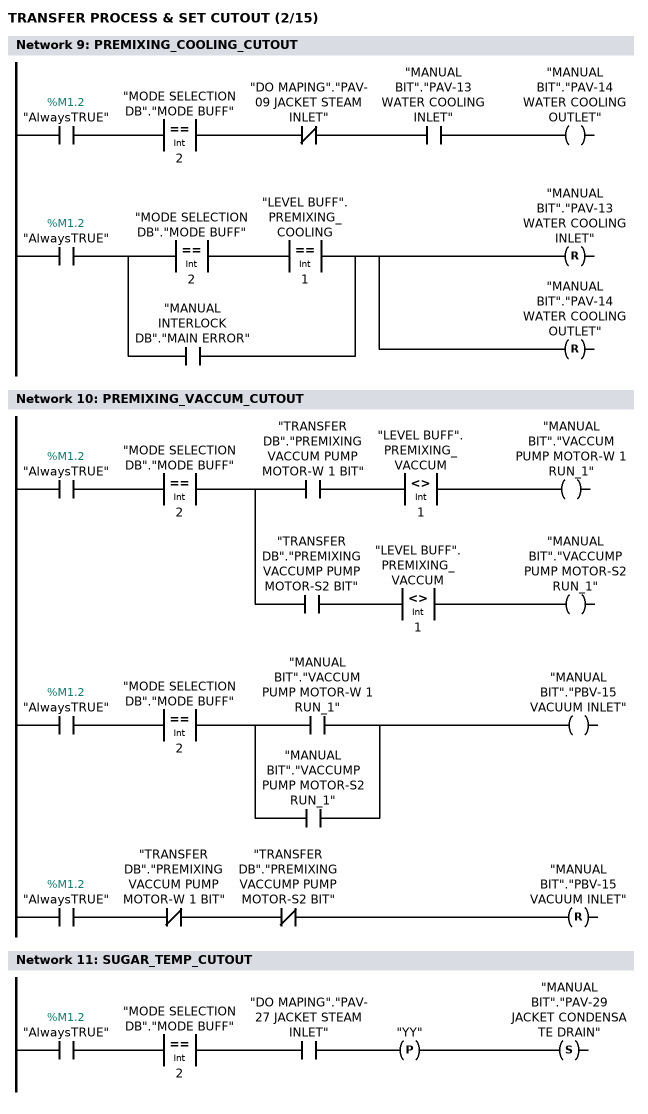
   RUNG wire#powerrail
      Contact( "AlwaysTRUE" )
      { S7_Templates := "SrcType := Int" } EQ_Contact(in1 := "MODE SELECTION DB"."MODE BUFF", in2 := 2)
      I_Contact( "DO MAPING"."PAV-09 JACKET STEAM INLET" )
      Contact( "MANUAL BIT"."PAV-13 WATER COOLING INLET" )
      Coil( "MANUAL BIT"."PAV-14 WATER COOLING OUTLET" )
   END_RUNG
   RUNG wire#powerrail
      Contact( "AlwaysTRUE" )
      wire#w1
      { S7_Templates := "SrcType := Int" } EQ_Contact(in1 := "MODE SELECTION DB"."MODE BUFF", in2 := 2)
      { S7_Templates := "SrcType := Int" } EQ_Contact(in1 := "LEVEL BUFF".PREMIXING_COOLING, in2 := 1)
      wire#w2
      R_Coil( "MANUAL BIT"."PAV-13 WATER COOLING INLET" )
   END_RUNG
   RUNG wire#w1
      Contact( "MANUAL INTERLOCK DB"."MAIN ERROR" )
   END_RUNG wire#w2
   RUNG wire#w2
      R_Coil( "MANUAL BIT"."PAV-14 WATER COOLING OUTLET" )
   END_RUNG
   // the same network as SCL:
   "MANUAL BIT"."PAV-14 WATER COOLING OUTLET" := "AlwaysTRUE" AND ("MODE SELECTION DB"."MODE BUFF" = 2) AND NOT "DO MAPING"."PAV-09 JACKET STEAM INLET" AND "MANUAL BIT"."PAV-13 WATER COOLING INLET";
   IF "AlwaysTRUE" AND ((("MODE SELECTION DB"."MODE BUFF" = 2) AND ("LEVEL BUFF".PREMIXING_COOLING = 1)) OR "MANUAL INTERLOCK DB"."MAIN ERROR") THEN
       "MANUAL BIT"."PAV-13 WATER COOLING INLET" := FALSE;
       "MANUAL BIT"."PAV-14 WATER COOLING OUTLET" := FALSE;
   END_IF;
END_REGION

REGION Network 10: PREMIXING_VACCUM_CUTOUT
   RUNG wire#powerrail
      Contact( "AlwaysTRUE" )
      { S7_Templates := "SrcType := Int" } EQ_Contact(in1 := "MODE SELECTION DB"."MODE BUFF", in2 := 2)
      wire#w1
      Contact( "TRANSFER DB"."PREMIXING VACCUM PUMP MOTOR-W 1 BIT" )
      { S7_Templates := "SrcType := Int" } NE_Contact(in1 := "LEVEL BUFF".PREMIXING_VACCUM, in2 := 1)
      Coil( "MANUAL BIT"."VACCUM PUMP MOTOR-W 1 RUN_1" )
   END_RUNG
   RUNG wire#w1
      Contact( "TRANSFER DB"."PREMIXING VACCUMP PUMP MOTOR-S2 BIT" )
      { S7_Templates := "SrcType := Int" } NE_Contact(in1 := "LEVEL BUFF".PREMIXING_VACCUM, in2 := 1)
      Coil( "MANUAL BIT"."VACCUMP PUMP MOTOR-S2 RUN_1" )
   END_RUNG
   RUNG wire#powerrail
      Contact( "AlwaysTRUE" )
      { S7_Templates := "SrcType := Int" } EQ_Contact(in1 := "MODE SELECTION DB"."MODE BUFF", in2 := 2)
      wire#w2
      Contact( "MANUAL BIT"."VACCUM PUMP MOTOR-W 1 RUN_1" )
      wire#w3
      Coil( "MANUAL BIT"."PBV-15 VACUUM INLET" )
   END_RUNG
   RUNG wire#w2
      Contact( "MANUAL BIT"."VACCUMP PUMP MOTOR-S2 RUN_1" )
   END_RUNG wire#w3
   RUNG wire#powerrail
      Contact( "AlwaysTRUE" )
      I_Contact( "TRANSFER DB"."PREMIXING VACCUM PUMP MOTOR-W 1 BIT" )
      I_Contact( "TRANSFER DB"."PREMIXING VACCUMP PUMP MOTOR-S2 BIT" )
      R_Coil( "MANUAL BIT"."PBV-15 VACUUM INLET" )
   END_RUNG
   // the same network as SCL:
   #_w1 := "AlwaysTRUE" AND ("MODE SELECTION DB"."MODE BUFF" = 2);
   "MANUAL BIT"."VACCUM PUMP MOTOR-W 1 RUN_1" := #_w1 AND "TRANSFER DB"."PREMIXING VACCUM PUMP MOTOR-W 1 BIT" AND ("LEVEL BUFF".PREMIXING_VACCUM <> 1);
   "MANUAL BIT"."VACCUMP PUMP MOTOR-S2 RUN_1" := #_w1 AND "TRANSFER DB"."PREMIXING VACCUMP PUMP MOTOR-S2 BIT" AND ("LEVEL BUFF".PREMIXING_VACCUM <> 1);
   "MANUAL BIT"."PBV-15 VACUUM INLET" := "AlwaysTRUE" AND ("MODE SELECTION DB"."MODE BUFF" = 2) AND ("MANUAL BIT"."VACCUM PUMP MOTOR-W 1 RUN_1" OR "MANUAL BIT"."VACCUMP PUMP MOTOR-S2 RUN_1");
   IF "AlwaysTRUE" AND NOT "TRANSFER DB"."PREMIXING VACCUM PUMP MOTOR-W 1 BIT" AND NOT "TRANSFER DB"."PREMIXING VACCUMP PUMP MOTOR-S2 BIT" THEN
       "MANUAL BIT"."PBV-15 VACUUM INLET" := FALSE;
   END_IF;
END_REGION

REGION Network 11: SUGAR_TEMP_CUTOUT
   RUNG wire#powerrail
      Contact( "AlwaysTRUE" )
      { S7_Templates := "SrcType := Int" } EQ_Contact(in1 := "MODE SELECTION DB"."MODE BUFF", in2 := 2)
      Contact( "DO MAPING"."PAV-27 JACKET STEAM INLET" )
      P_Trig( "YY" )
      S_Coil( "MANUAL BIT"."PAV-29 JACKET CONDENSATE DRAIN" )
   END_RUNG
   // the same network as SCL:
   #_w1 := "AlwaysTRUE" AND ("MODE SELECTION DB"."MODE BUFF" = 2) AND "DO MAPING"."PAV-27 JACKET STEAM INLET";
   #_w2 := #_w1 AND NOT "YY";   // rising edge
   "YY" := #_w1;
   IF #_w2 THEN "MANUAL BIT"."PAV-29 JACKET CONDENSATE DRAIN" := TRUE; END_IF;
END_REGION

REGION Network 12: SUGAR_VACCUM_CUTOUT
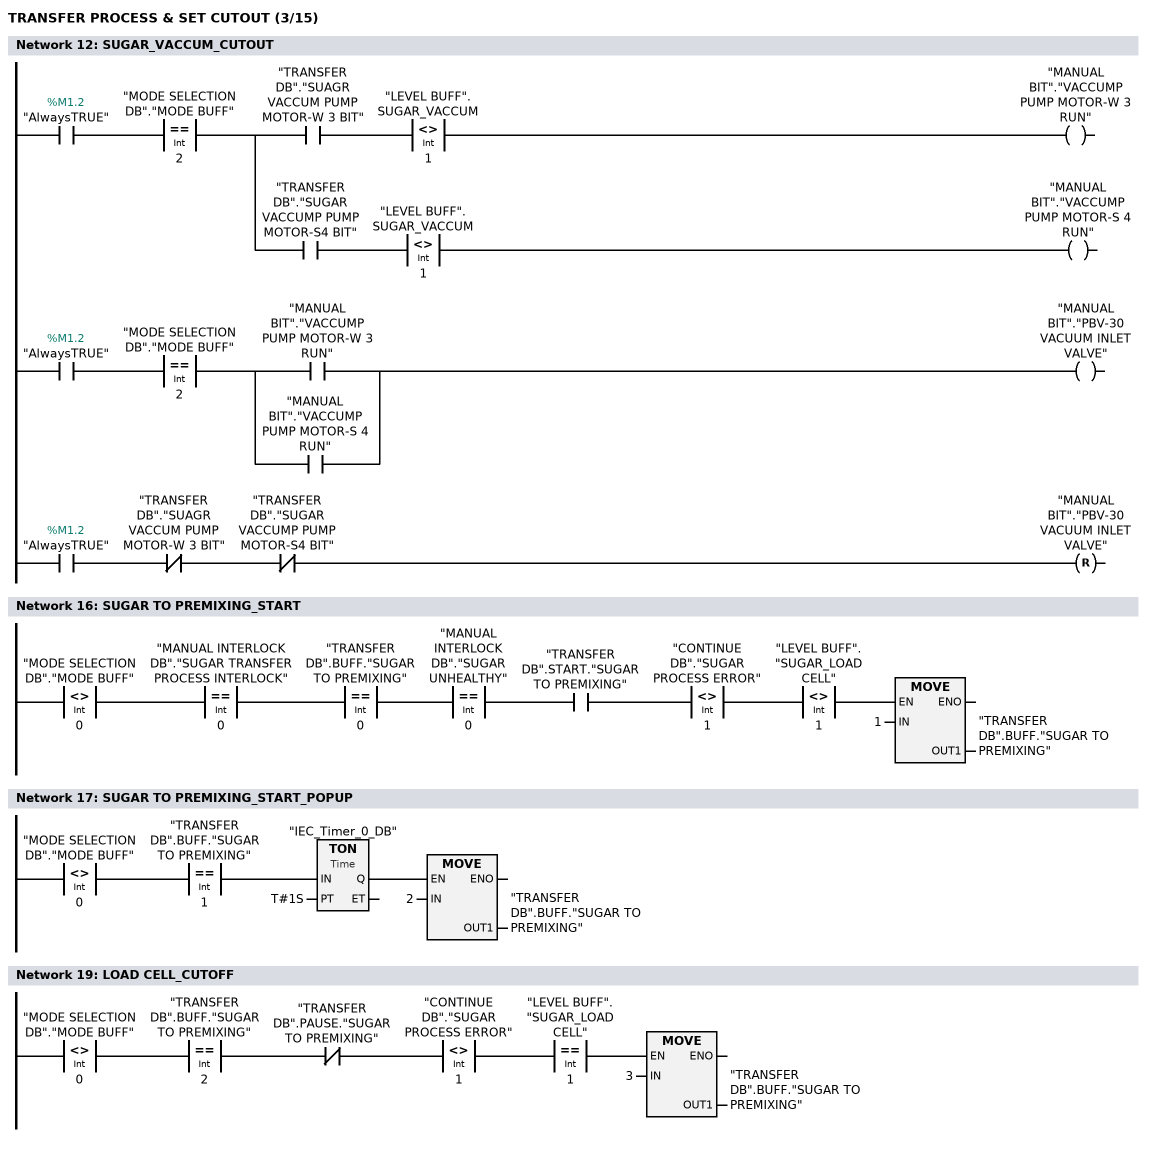
   RUNG wire#powerrail
      Contact( "AlwaysTRUE" )
      { S7_Templates := "SrcType := Int" } EQ_Contact(in1 := "MODE SELECTION DB"."MODE BUFF", in2 := 2)
      wire#w1
      Contact( "TRANSFER DB"."SUAGR VACCUM PUMP MOTOR-W 3 BIT" )
      { S7_Templates := "SrcType := Int" } NE_Contact(in1 := "LEVEL BUFF".SUGAR_VACCUM, in2 := 1)
      Coil( "MANUAL BIT"."VACCUMP PUMP MOTOR-W 3 RUN" )
   END_RUNG
   RUNG wire#w1
      Contact( "TRANSFER DB"."SUGAR VACCUMP PUMP MOTOR-S4 BIT" )
      { S7_Templates := "SrcType := Int" } NE_Contact(in1 := "LEVEL BUFF".SUGAR_VACCUM, in2 := 1)
      Coil( "MANUAL BIT"."VACCUMP PUMP MOTOR-S 4 RUN" )
   END_RUNG
   RUNG wire#powerrail
      Contact( "AlwaysTRUE" )
      { S7_Templates := "SrcType := Int" } EQ_Contact(in1 := "MODE SELECTION DB"."MODE BUFF", in2 := 2)
      wire#w2
      Contact( "MANUAL BIT"."VACCUMP PUMP MOTOR-W 3 RUN" )
      wire#w3
      Coil( "MANUAL BIT"."PBV-30 VACUUM INLET VALVE" )
   END_RUNG
   RUNG wire#w2
      Contact( "MANUAL BIT"."VACCUMP PUMP MOTOR-S 4 RUN" )
   END_RUNG wire#w3
   RUNG wire#powerrail
      Contact( "AlwaysTRUE" )
      I_Contact( "TRANSFER DB"."SUAGR VACCUM PUMP MOTOR-W 3 BIT" )
      I_Contact( "TRANSFER DB"."SUGAR VACCUMP PUMP MOTOR-S4 BIT" )
      R_Coil( "MANUAL BIT"."PBV-30 VACUUM INLET VALVE" )
   END_RUNG
   // the same network as SCL:
   #_w1 := "AlwaysTRUE" AND ("MODE SELECTION DB"."MODE BUFF" = 2);
   "MANUAL BIT"."VACCUMP PUMP MOTOR-W 3 RUN" := #_w1 AND "TRANSFER DB"."SUAGR VACCUM PUMP MOTOR-W 3 BIT" AND ("LEVEL BUFF".SUGAR_VACCUM <> 1);
   "MANUAL BIT"."VACCUMP PUMP MOTOR-S 4 RUN" := #_w1 AND "TRANSFER DB"."SUGAR VACCUMP PUMP MOTOR-S4 BIT" AND ("LEVEL BUFF".SUGAR_VACCUM <> 1);
   "MANUAL BIT"."PBV-30 VACUUM INLET VALVE" := "AlwaysTRUE" AND ("MODE SELECTION DB"."MODE BUFF" = 2) AND ("MANUAL BIT"."VACCUMP PUMP MOTOR-W 3 RUN" OR "MANUAL BIT"."VACCUMP PUMP MOTOR-S 4 RUN");
   IF "AlwaysTRUE" AND NOT "TRANSFER DB"."SUAGR VACCUM PUMP MOTOR-W 3 BIT" AND NOT "TRANSFER DB"."SUGAR VACCUMP PUMP MOTOR-S4 BIT" THEN
       "MANUAL BIT"."PBV-30 VACUUM INLET VALVE" := FALSE;
   END_IF;
END_REGION

REGION Network 15: ////////////////////////////////////////////////////////////////////// TRANSFER PROCESS- SUGAR //////////////////////////////////////////////////////////////////////////////////
END_REGION

REGION Network 16: SUGAR TO PREMIXING_START
   RUNG wire#powerrail
      { S7_Templates := "SrcType := Int" } NE_Contact(in1 := "MODE SELECTION DB"."MODE BUFF", in2 := 0)
      { S7_Templates := "SrcType := Int" } EQ_Contact(in1 := "MANUAL INTERLOCK DB"."SUGAR TRANSFER PROCESS INTERLOCK", in2 := 0)
      { S7_Templates := "SrcType := Int" } EQ_Contact(in1 := "TRANSFER DB".BUFF."SUGAR TO PREMIXING", in2 := 0)
      { S7_Templates := "SrcType := Int" } EQ_Contact(in1 := "MANUAL INTERLOCK DB"."SUGAR UNHEALTHY", in2 := 0)
      Contact( "TRANSFER DB".START."SUGAR TO PREMIXING" )
      { S7_Templates := "SrcType := Int" } NE_Contact(in1 := "CONTINUE DB"."SUGAR PROCESS ERROR", in2 := 1)
      { S7_Templates := "SrcType := Int" } NE_Contact(in1 := "LEVEL BUFF"."SUGAR_LOAD CELL", in2 := 1)
      Move(in := 1, out1 => "TRANSFER DB".BUFF."SUGAR TO PREMIXING")
   END_RUNG
   // the same network as SCL:
   IF ("MODE SELECTION DB"."MODE BUFF" <> 0) AND ("MANUAL INTERLOCK DB"."SUGAR TRANSFER PROCESS INTERLOCK" = 0) AND ("TRANSFER DB".BUFF."SUGAR TO PREMIXING" = 0) AND ("MANUAL INTERLOCK DB"."SUGAR UNHEALTHY" = 0) AND "TRANSFER DB".START."SUGAR TO PREMIXING" AND ("CONTINUE DB"."SUGAR PROCESS ERROR" <> 1) AND ("LEVEL BUFF"."SUGAR_LOAD CELL" <> 1) THEN
       "TRANSFER DB".BUFF."SUGAR TO PREMIXING" := 1;
   END_IF;
END_REGION

REGION Network 17: SUGAR TO PREMIXING_START_POPUP
   RUNG wire#powerrail
      { S7_Templates := "SrcType := Int" } NE_Contact(in1 := "MODE SELECTION DB"."MODE BUFF", in2 := 0)
      { S7_Templates := "SrcType := Int" } EQ_Contact(in1 := "TRANSFER DB".BUFF."SUGAR TO PREMIXING", in2 := 1)
      { S7_Templates := "time_type := Time" } "IEC_Timer_0_DB".TON(pt := T#1S, et =>)
      Move(in := 2, out1 => "TRANSFER DB".BUFF."SUGAR TO PREMIXING")
   END_RUNG
   // the same network as SCL:
   "IEC_Timer_0_DB".TON(IN := ("MODE SELECTION DB"."MODE BUFF" <> 0) AND ("TRANSFER DB".BUFF."SUGAR TO PREMIXING" = 1),
                        PT := T#1S);
   IF "IEC_Timer_0_DB".Q THEN "TRANSFER DB".BUFF."SUGAR TO PREMIXING" := 2; END_IF;
END_REGION

REGION Network 18 (SCL): OPENVALVE
   IF "MODE SELECTION DB"."MODE BUFF" <> 0 AND "TRANSFER DB".BUFF."SUGAR TO PREMIXING" = 2
       AND NOT "TRANSFER DB".PAUSE."SUGAR TO PREMIXING" AND
       "CONTINUE DB"."SUGAR PROCESS ERROR" = 0 AND "LEVEL BUFF"."SUGAR_LOAD CELL" = 0 THEN
       "TRANSFER DB".BIT."SUGAR TO PREMIXING"."PFBV-32 TANK OUTLET VALVE" := TRUE;
       "TRANSFER DB".BIT."SUGAR TO PREMIXING"."PBV-80 BOTTOM OUTLET TO BASKET FILTER" := TRUE;
       "TRANSFER DB".BIT."SUGAR TO PREMIXING"."BASKET FILTER MOTOR RUN" := TRUE;
       "TRANSFER DB".BIT."SUGAR TO PREMIXING"."PBV-79 BASKET FILTER INLET" := TRUE;
       "TRANSFER DB".BIT."SUGAR TO PREMIXING"."PBV-149" := TRUE;
       "TRANSFER DB".BIT."SUGAR TO PREMIXING"."PBV-88 BASKET FILTER TRANSFER LINE" := TRUE;
       "TRANSFER DB".BIT."SUGAR TO PREMIXING"."PBV-87 BASKET FILTER TO PREMIX VESSEL LINE" := TRUE;
   ELSE
       "TRANSFER DB".BIT."SUGAR TO PREMIXING"."PFBV-32 TANK OUTLET VALVE" := FALSE;
       "TRANSFER DB".BIT."SUGAR TO PREMIXING"."PBV-80 BOTTOM OUTLET TO BASKET FILTER" := FALSE;
       "TRANSFER DB".BIT."SUGAR TO PREMIXING"."BASKET FILTER MOTOR RUN" := FALSE;
       "TRANSFER DB".BIT."SUGAR TO PREMIXING"."PBV-79 BASKET FILTER INLET" := FALSE;
       "TRANSFER DB".BIT."SUGAR TO PREMIXING"."PBV-149" := FALSE;
       "TRANSFER DB".BIT."SUGAR TO PREMIXING"."PBV-88 BASKET FILTER TRANSFER LINE" := FALSE;
       "TRANSFER DB".BIT."SUGAR TO PREMIXING"."PBV-87 BASKET FILTER TO PREMIX VESSEL LINE" := FALSE;
       ;
   END_IF;
END_REGION

REGION Network 19: LOAD CELL_CUTOFF
   RUNG wire#powerrail
      { S7_Templates := "SrcType := Int" } NE_Contact(in1 := "MODE SELECTION DB"."MODE BUFF", in2 := 0)
      { S7_Templates := "SrcType := Int" } EQ_Contact(in1 := "TRANSFER DB".BUFF."SUGAR TO PREMIXING", in2 := 2)
      I_Contact( "TRANSFER DB".PAUSE."SUGAR TO PREMIXING" )
      { S7_Templates := "SrcType := Int" } NE_Contact(in1 := "CONTINUE DB"."SUGAR PROCESS ERROR", in2 := 1)
      { S7_Templates := "SrcType := Int" } EQ_Contact(in1 := "LEVEL BUFF"."SUGAR_LOAD CELL", in2 := 1)
      Move(in := 3, out1 => "TRANSFER DB".BUFF."SUGAR TO PREMIXING")
   END_RUNG
   // the same network as SCL:
   IF ("MODE SELECTION DB"."MODE BUFF" <> 0) AND ("TRANSFER DB".BUFF."SUGAR TO PREMIXING" = 2) AND NOT "TRANSFER DB".PAUSE."SUGAR TO PREMIXING" AND ("CONTINUE DB"."SUGAR PROCESS ERROR" <> 1) AND ("LEVEL BUFF"."SUGAR_LOAD CELL" = 1) THEN
       "TRANSFER DB".BUFF."SUGAR TO PREMIXING" := 3;
   END_IF;
END_REGION

REGION Network 20: PROCESS OVER & STOP
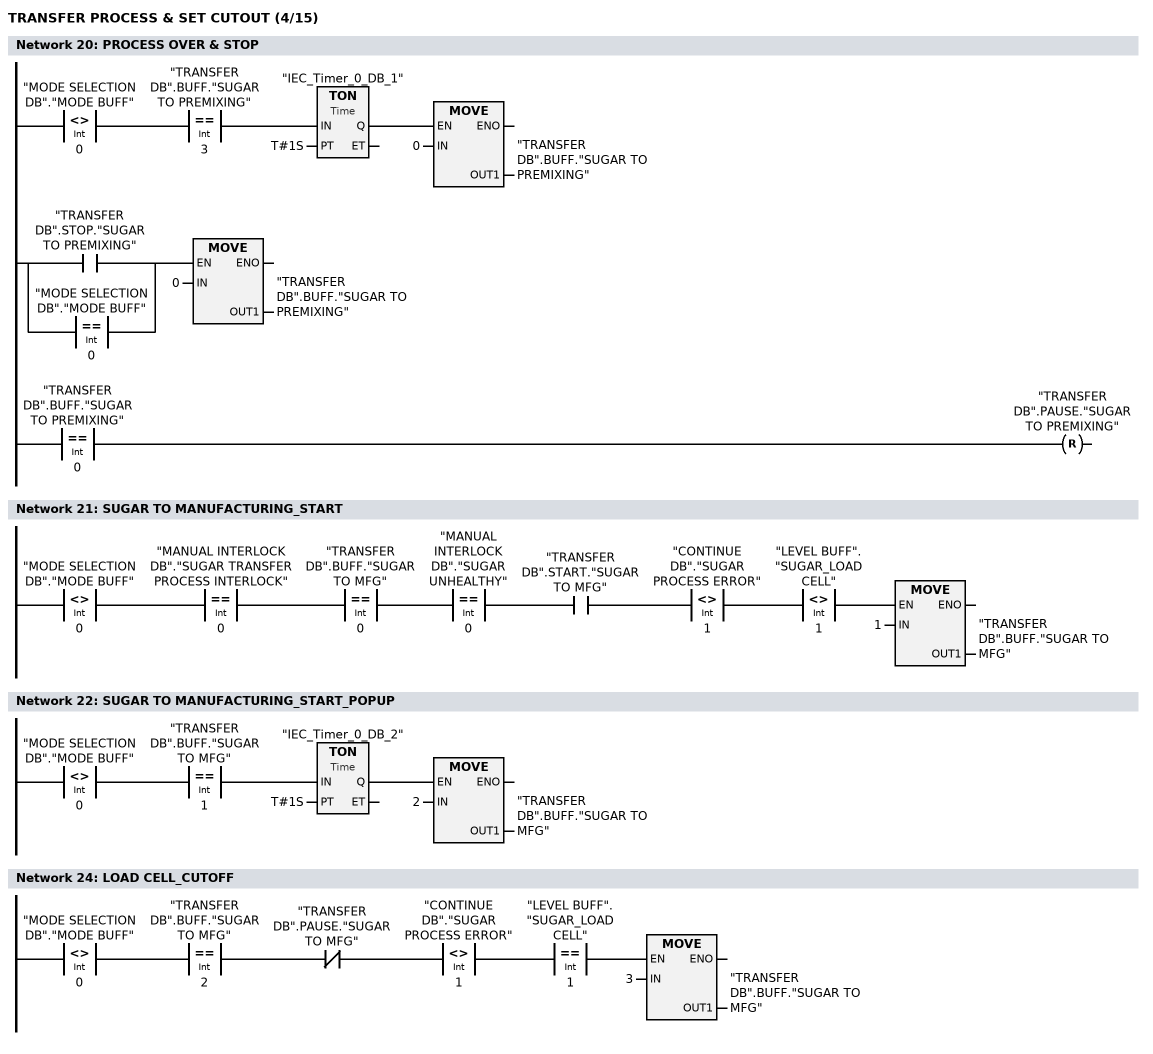
   RUNG wire#powerrail
      { S7_Templates := "SrcType := Int" } NE_Contact(in1 := "MODE SELECTION DB"."MODE BUFF", in2 := 0)
      { S7_Templates := "SrcType := Int" } EQ_Contact(in1 := "TRANSFER DB".BUFF."SUGAR TO PREMIXING", in2 := 3)
      { S7_Templates := "time_type := Time" } "IEC_Timer_0_DB_1".TON(pt := T#1S, et =>)
      Move(in := 0, out1 => "TRANSFER DB".BUFF."SUGAR TO PREMIXING")
   END_RUNG
   RUNG wire#powerrail
      Contact( "TRANSFER DB".STOP."SUGAR TO PREMIXING" )
      wire#w1
      Move(in := 0, out1 => "TRANSFER DB".BUFF."SUGAR TO PREMIXING")
   END_RUNG
   RUNG wire#powerrail
      { S7_Templates := "SrcType := Int" } EQ_Contact(in1 := "MODE SELECTION DB"."MODE BUFF", in2 := 0)
   END_RUNG wire#w1
   RUNG wire#powerrail
      { S7_Templates := "SrcType := Int" } EQ_Contact(in1 := "TRANSFER DB".BUFF."SUGAR TO PREMIXING", in2 := 0)
      R_Coil( "TRANSFER DB".PAUSE."SUGAR TO PREMIXING" )
   END_RUNG
   // the same network as SCL:
   "IEC_Timer_0_DB_1".TON(IN := ("MODE SELECTION DB"."MODE BUFF" <> 0) AND ("TRANSFER DB".BUFF."SUGAR TO PREMIXING" = 3),
                          PT := T#1S);
   IF "IEC_Timer_0_DB_1".Q THEN "TRANSFER DB".BUFF."SUGAR TO PREMIXING" := 0; END_IF;
   IF "TRANSFER DB".STOP."SUGAR TO PREMIXING" OR ("MODE SELECTION DB"."MODE BUFF" = 0) THEN
       "TRANSFER DB".BUFF."SUGAR TO PREMIXING" := 0;
   END_IF;
   IF "TRANSFER DB".BUFF."SUGAR TO PREMIXING" = 0 THEN
       "TRANSFER DB".PAUSE."SUGAR TO PREMIXING" := FALSE;
   END_IF;
END_REGION

REGION Network 21: SUGAR TO MANUFACTURING_START
   RUNG wire#powerrail
      { S7_Templates := "SrcType := Int" } NE_Contact(in1 := "MODE SELECTION DB"."MODE BUFF", in2 := 0)
      { S7_Templates := "SrcType := Int" } EQ_Contact(in1 := "MANUAL INTERLOCK DB"."SUGAR TRANSFER PROCESS INTERLOCK", in2 := 0)
      { S7_Templates := "SrcType := Int" } EQ_Contact(in1 := "TRANSFER DB".BUFF."SUGAR TO MFG", in2 := 0)
      { S7_Templates := "SrcType := Int" } EQ_Contact(in1 := "MANUAL INTERLOCK DB"."SUGAR UNHEALTHY", in2 := 0)
      Contact( "TRANSFER DB".START."SUGAR TO MFG" )
      { S7_Templates := "SrcType := Int" } NE_Contact(in1 := "CONTINUE DB"."SUGAR PROCESS ERROR", in2 := 1)
      { S7_Templates := "SrcType := Int" } NE_Contact(in1 := "LEVEL BUFF"."SUGAR_LOAD CELL", in2 := 1)
      Move(in := 1, out1 => "TRANSFER DB".BUFF."SUGAR TO MFG")
   END_RUNG
   // the same network as SCL:
   IF ("MODE SELECTION DB"."MODE BUFF" <> 0) AND ("MANUAL INTERLOCK DB"."SUGAR TRANSFER PROCESS INTERLOCK" = 0) AND ("TRANSFER DB".BUFF."SUGAR TO MFG" = 0) AND ("MANUAL INTERLOCK DB"."SUGAR UNHEALTHY" = 0) AND "TRANSFER DB".START."SUGAR TO MFG" AND ("CONTINUE DB"."SUGAR PROCESS ERROR" <> 1) AND ("LEVEL BUFF"."SUGAR_LOAD CELL" <> 1) THEN
       "TRANSFER DB".BUFF."SUGAR TO MFG" := 1;
   END_IF;
END_REGION

REGION Network 22: SUGAR TO MANUFACTURING_START_POPUP
   RUNG wire#powerrail
      { S7_Templates := "SrcType := Int" } NE_Contact(in1 := "MODE SELECTION DB"."MODE BUFF", in2 := 0)
      { S7_Templates := "SrcType := Int" } EQ_Contact(in1 := "TRANSFER DB".BUFF."SUGAR TO MFG", in2 := 1)
      { S7_Templates := "time_type := Time" } "IEC_Timer_0_DB_2".TON(pt := T#1S, et =>)
      Move(in := 2, out1 => "TRANSFER DB".BUFF."SUGAR TO MFG")
   END_RUNG
   // the same network as SCL:
   "IEC_Timer_0_DB_2".TON(IN := ("MODE SELECTION DB"."MODE BUFF" <> 0) AND ("TRANSFER DB".BUFF."SUGAR TO MFG" = 1),
                          PT := T#1S);
   IF "IEC_Timer_0_DB_2".Q THEN "TRANSFER DB".BUFF."SUGAR TO MFG" := 2; END_IF;
END_REGION

REGION Network 23 (SCL): OPENVALVE
   IF "MODE SELECTION DB"."MODE BUFF" <> 0 AND "TRANSFER DB".BUFF."SUGAR TO MFG" = 2
       AND NOT "TRANSFER DB".PAUSE."SUGAR TO MFG" 
       AND "CONTINUE DB"."SUGAR PROCESS ERROR" = 0 AND "LEVEL BUFF"."SUGAR_LOAD CELL" = 0 THEN
       "TRANSFER DB".BIT."SUGAR TO MFG"."PFBV-32 TANK OUTLET VALVE" := TRUE;
       "TRANSFER DB".BIT."SUGAR TO MFG"."PBV-80 BOTTOM OUTLET TO BASKET FILTER" := TRUE;
       "TRANSFER DB".BIT."SUGAR TO MFG"."BASKET FILTER MOTOR RUN" := TRUE;
       "TRANSFER DB".BIT."SUGAR TO MFG"."PBV-79 BASKET FILTER INLET" := TRUE;
       "TRANSFER DB".BIT."SUGAR TO MFG"."PBV-149" := TRUE;
       "TRANSFER DB".BIT."SUGAR TO MFG"."PBV-89 BASKET FILTER TO MFG INLET TRANSFER LINE" := TRUE;
       "TRANSFER DB".BIT."SUGAR TO MFG"."PBV-101 SUGAR MELTING TO MFG TRANSFER (TOP DISH)" := TRUE;

   ELSE
       "TRANSFER DB".BIT."SUGAR TO MFG"."PFBV-32 TANK OUTLET VALVE" := FALSE;
       "TRANSFER DB".BIT."SUGAR TO MFG"."PBV-80 BOTTOM OUTLET TO BASKET FILTER" := FALSE;
       "TRANSFER DB".BIT."SUGAR TO MFG"."BASKET FILTER MOTOR RUN" := FALSE;
       "TRANSFER DB".BIT."SUGAR TO MFG"."PBV-79 BASKET FILTER INLET" := FALSE;
       "TRANSFER DB".BIT."SUGAR TO MFG"."PBV-149" := FALSE;
       "TRANSFER DB".BIT."SUGAR TO MFG"."PBV-89 BASKET FILTER TO MFG INLET TRANSFER LINE" := FALSE;
       "TRANSFER DB".BIT."SUGAR TO MFG"."PBV-101 SUGAR MELTING TO MFG TRANSFER (TOP DISH)" := FALSE;
       ;
   END_IF;
END_REGION

REGION Network 24: LOAD CELL_CUTOFF
   RUNG wire#powerrail
      { S7_Templates := "SrcType := Int" } NE_Contact(in1 := "MODE SELECTION DB"."MODE BUFF", in2 := 0)
      { S7_Templates := "SrcType := Int" } EQ_Contact(in1 := "TRANSFER DB".BUFF."SUGAR TO MFG", in2 := 2)
      I_Contact( "TRANSFER DB".PAUSE."SUGAR TO MFG" )
      { S7_Templates := "SrcType := Int" } NE_Contact(in1 := "CONTINUE DB"."SUGAR PROCESS ERROR", in2 := 1)
      { S7_Templates := "SrcType := Int" } EQ_Contact(in1 := "LEVEL BUFF"."SUGAR_LOAD CELL", in2 := 1)
      Move(in := 3, out1 => "TRANSFER DB".BUFF."SUGAR TO MFG")
   END_RUNG
   // the same network as SCL:
   IF ("MODE SELECTION DB"."MODE BUFF" <> 0) AND ("TRANSFER DB".BUFF."SUGAR TO MFG" = 2) AND NOT "TRANSFER DB".PAUSE."SUGAR TO MFG" AND ("CONTINUE DB"."SUGAR PROCESS ERROR" <> 1) AND ("LEVEL BUFF"."SUGAR_LOAD CELL" = 1) THEN
       "TRANSFER DB".BUFF."SUGAR TO MFG" := 3;
   END_IF;
END_REGION

REGION Network 25: PROCESS OVER & STOP
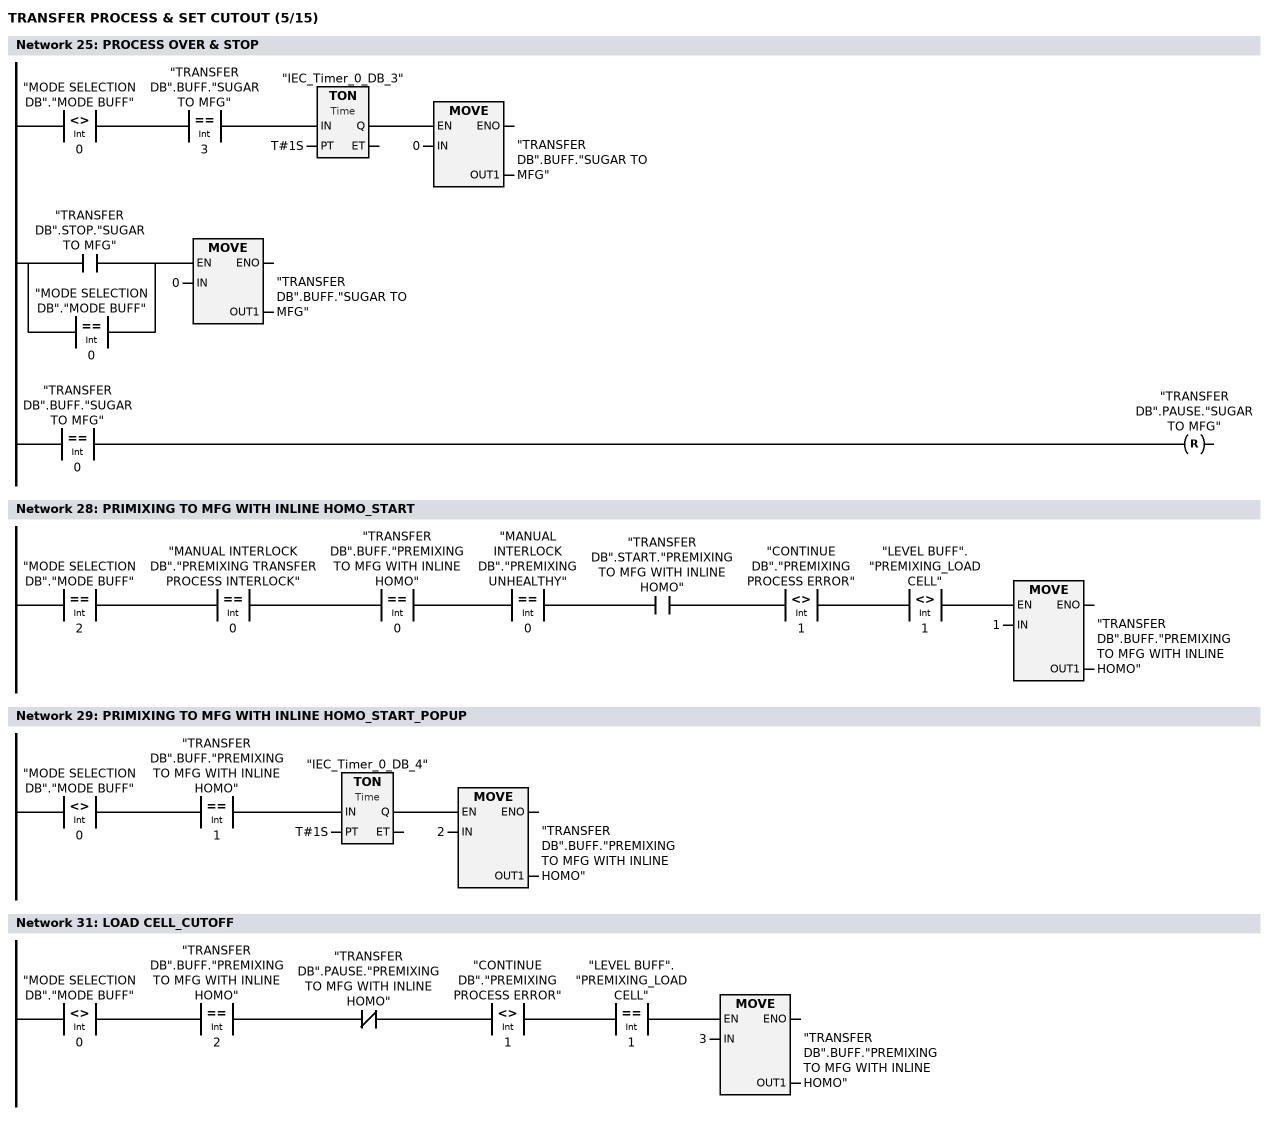
   RUNG wire#powerrail
      { S7_Templates := "SrcType := Int" } NE_Contact(in1 := "MODE SELECTION DB"."MODE BUFF", in2 := 0)
      { S7_Templates := "SrcType := Int" } EQ_Contact(in1 := "TRANSFER DB".BUFF."SUGAR TO MFG", in2 := 3)
      { S7_Templates := "time_type := Time" } "IEC_Timer_0_DB_3".TON(pt := T#1S, et =>)
      Move(in := 0, out1 => "TRANSFER DB".BUFF."SUGAR TO MFG")
   END_RUNG
   RUNG wire#powerrail
      Contact( "TRANSFER DB".STOP."SUGAR TO MFG" )
      wire#w1
      Move(in := 0, out1 => "TRANSFER DB".BUFF."SUGAR TO MFG")
   END_RUNG
   RUNG wire#powerrail
      { S7_Templates := "SrcType := Int" } EQ_Contact(in1 := "MODE SELECTION DB"."MODE BUFF", in2 := 0)
   END_RUNG wire#w1
   RUNG wire#powerrail
      { S7_Templates := "SrcType := Int" } EQ_Contact(in1 := "TRANSFER DB".BUFF."SUGAR TO MFG", in2 := 0)
      R_Coil( "TRANSFER DB".PAUSE."SUGAR TO MFG" )
   END_RUNG
   // the same network as SCL:
   "IEC_Timer_0_DB_3".TON(IN := ("MODE SELECTION DB"."MODE BUFF" <> 0) AND ("TRANSFER DB".BUFF."SUGAR TO MFG" = 3),
                          PT := T#1S);
   IF "IEC_Timer_0_DB_3".Q THEN "TRANSFER DB".BUFF."SUGAR TO MFG" := 0; END_IF;
   IF "TRANSFER DB".STOP."SUGAR TO MFG" OR ("MODE SELECTION DB"."MODE BUFF" = 0) THEN
       "TRANSFER DB".BUFF."SUGAR TO MFG" := 0;
   END_IF;
   IF "TRANSFER DB".BUFF."SUGAR TO MFG" = 0 THEN "TRANSFER DB".PAUSE."SUGAR TO MFG" := FALSE; END_IF;
END_REGION

REGION Network 27: ////////////////////////////////////////////////////////////////////// TRANSFER PROCESS- PREMIXING //////////////////////////////////////////////////////////////////////////////////
END_REGION

REGION Network 28: PRIMIXING TO MFG WITH INLINE HOMO_START
   RUNG wire#powerrail
      { S7_Templates := "SrcType := Int" } EQ_Contact(in1 := "MODE SELECTION DB"."MODE BUFF", in2 := 2)
      { S7_Templates := "SrcType := Int" } EQ_Contact(in1 := "MANUAL INTERLOCK DB"."PREMIXING TRANSFER PROCESS INTERLOCK", in2 := 0)
      { S7_Templates := "SrcType := Int" } EQ_Contact(in1 := "TRANSFER DB".BUFF."PREMIXING TO MFG WITH INLINE HOMO", in2 := 0)
      { S7_Templates := "SrcType := Int" } EQ_Contact(in1 := "MANUAL INTERLOCK DB"."PREMIXING UNHEALTHY", in2 := 0)
      Contact( "TRANSFER DB".START."PREMIXING TO MFG WITH INLINE HOMO" )
      { S7_Templates := "SrcType := Int" } NE_Contact(in1 := "CONTINUE DB"."PREMIXING PROCESS ERROR", in2 := 1)
      { S7_Templates := "SrcType := Int" } NE_Contact(in1 := "LEVEL BUFF"."PREMIXING_LOAD CELL", in2 := 1)
      Move(in := 1, out1 => "TRANSFER DB".BUFF."PREMIXING TO MFG WITH INLINE HOMO")
   END_RUNG
   // the same network as SCL:
   IF ("MODE SELECTION DB"."MODE BUFF" = 2) AND ("MANUAL INTERLOCK DB"."PREMIXING TRANSFER PROCESS INTERLOCK" = 0) AND ("TRANSFER DB".BUFF."PREMIXING TO MFG WITH INLINE HOMO" = 0) AND ("MANUAL INTERLOCK DB"."PREMIXING UNHEALTHY" = 0) AND "TRANSFER DB".START."PREMIXING TO MFG WITH INLINE HOMO" AND ("CONTINUE DB"."PREMIXING PROCESS ERROR" <> 1) AND ("LEVEL BUFF"."PREMIXING_LOAD CELL" <> 1) THEN
       "TRANSFER DB".BUFF."PREMIXING TO MFG WITH INLINE HOMO" := 1;
   END_IF;
END_REGION

REGION Network 29: PRIMIXING TO MFG WITH INLINE HOMO_START_POPUP
   RUNG wire#powerrail
      { S7_Templates := "SrcType := Int" } NE_Contact(in1 := "MODE SELECTION DB"."MODE BUFF", in2 := 0)
      { S7_Templates := "SrcType := Int" } EQ_Contact(in1 := "TRANSFER DB".BUFF."PREMIXING TO MFG WITH INLINE HOMO", in2 := 1)
      { S7_Templates := "time_type := Time" } "IEC_Timer_0_DB_4".TON(pt := T#1S, et =>)
      Move(in := 2, out1 => "TRANSFER DB".BUFF."PREMIXING TO MFG WITH INLINE HOMO")
   END_RUNG
   // the same network as SCL:
   "IEC_Timer_0_DB_4".TON(IN := ("MODE SELECTION DB"."MODE BUFF" <> 0) AND ("TRANSFER DB".BUFF."PREMIXING TO MFG WITH INLINE HOMO" = 1),
                          PT := T#1S);
   IF "IEC_Timer_0_DB_4".Q THEN "TRANSFER DB".BUFF."PREMIXING TO MFG WITH INLINE HOMO" := 2; END_IF;
END_REGION

REGION Network 30 (SCL): OPENVALVE
   IF "MODE SELECTION DB"."MODE BUFF" <> 0 AND "TRANSFER DB".BUFF."PREMIXING TO MFG WITH INLINE HOMO" = 2
       AND NOT "TRANSFER DB".PAUSE."PREMIXING TO MFG WITH INLINE HOMO" 
       AND "CONTINUE DB"."PREMIXING PROCESS ERROR" = 0 AND "LEVEL BUFF"."PREMIXING_LOAD CELL" = 0 THEN
       "TRANSFER DB".BIT."PREMIXING TO MFG WITH INLINE HOMO"."PFBV-17 TANK OUTLET VALVE" := TRUE;
       "TRANSFER DB".BIT."PREMIXING TO MFG WITH INLINE HOMO"."PBV-93 TANK OUTLET TO INLINE HOMOGENIZER LINE" := TRUE;
       "TRANSFER DB".BIT."PREMIXING TO MFG WITH INLINE HOMO"."PBV-94 INLINE HOMOGENIZER INLET LINE" := TRUE;
       "TRANSFER DB".BIT."PREMIXING TO MFG WITH INLINE HOMO"."INLINE 2 HOMOGENIZER MOTOR 2 RUN" := TRUE;
       "TRANSFER DB".BIT."PREMIXING TO MFG WITH INLINE HOMO"."PBV-96 INLINE HOMOGENIZER RECIRCULATION LINE" := TRUE;
       "TRANSFER DB".BIT."PREMIXING TO MFG WITH INLINE HOMO"."PBV-91 PREMIX TO MFG TRANSFER LINE" := TRUE;
       "TRANSFER DB".BIT."PREMIXING TO MFG WITH INLINE HOMO"."PBV-102 PREMIX TO MFG TRANSFER (TOP DISH)" := TRUE;

   ELSE
       "TRANSFER DB".BIT."PREMIXING TO MFG WITH INLINE HOMO"."PFBV-17 TANK OUTLET VALVE" := FALSE;
       "TRANSFER DB".BIT."PREMIXING TO MFG WITH INLINE HOMO"."PBV-93 TANK OUTLET TO INLINE HOMOGENIZER LINE" := FALSE;
       "TRANSFER DB".BIT."PREMIXING TO MFG WITH INLINE HOMO"."PBV-94 INLINE HOMOGENIZER INLET LINE" := FALSE;
       "TRANSFER DB".BIT."PREMIXING TO MFG WITH INLINE HOMO"."INLINE 2 HOMOGENIZER MOTOR 2 RUN" := FALSE;
       "TRANSFER DB".BIT."PREMIXING TO MFG WITH INLINE HOMO"."PBV-96 INLINE HOMOGENIZER RECIRCULATION LINE" := FALSE;
       "TRANSFER DB".BIT."PREMIXING TO MFG WITH INLINE HOMO"."PBV-91 PREMIX TO MFG TRANSFER LINE" := FALSE;
       "TRANSFER DB".BIT."PREMIXING TO MFG WITH INLINE HOMO"."PBV-102 PREMIX TO MFG TRANSFER (TOP DISH)" := FALSE;
       ;
   END_IF;
END_REGION

REGION Network 31: LOAD CELL_CUTOFF
   RUNG wire#powerrail
      { S7_Templates := "SrcType := Int" } NE_Contact(in1 := "MODE SELECTION DB"."MODE BUFF", in2 := 0)
      { S7_Templates := "SrcType := Int" } EQ_Contact(in1 := "TRANSFER DB".BUFF."PREMIXING TO MFG WITH INLINE HOMO", in2 := 2)
      I_Contact( "TRANSFER DB".PAUSE."PREMIXING TO MFG WITH INLINE HOMO" )
      { S7_Templates := "SrcType := Int" } NE_Contact(in1 := "CONTINUE DB"."PREMIXING PROCESS ERROR", in2 := 1)
      { S7_Templates := "SrcType := Int" } EQ_Contact(in1 := "LEVEL BUFF"."PREMIXING_LOAD CELL", in2 := 1)
      Move(in := 3, out1 => "TRANSFER DB".BUFF."PREMIXING TO MFG WITH INLINE HOMO")
   END_RUNG
   // the same network as SCL:
   IF ("MODE SELECTION DB"."MODE BUFF" <> 0) AND ("TRANSFER DB".BUFF."PREMIXING TO MFG WITH INLINE HOMO" = 2) AND NOT "TRANSFER DB".PAUSE."PREMIXING TO MFG WITH INLINE HOMO" AND ("CONTINUE DB"."PREMIXING PROCESS ERROR" <> 1) AND ("LEVEL BUFF"."PREMIXING_LOAD CELL" = 1) THEN
       "TRANSFER DB".BUFF."PREMIXING TO MFG WITH INLINE HOMO" := 3;
   END_IF;
END_REGION

REGION Network 32: PROCESS OVER & STOP
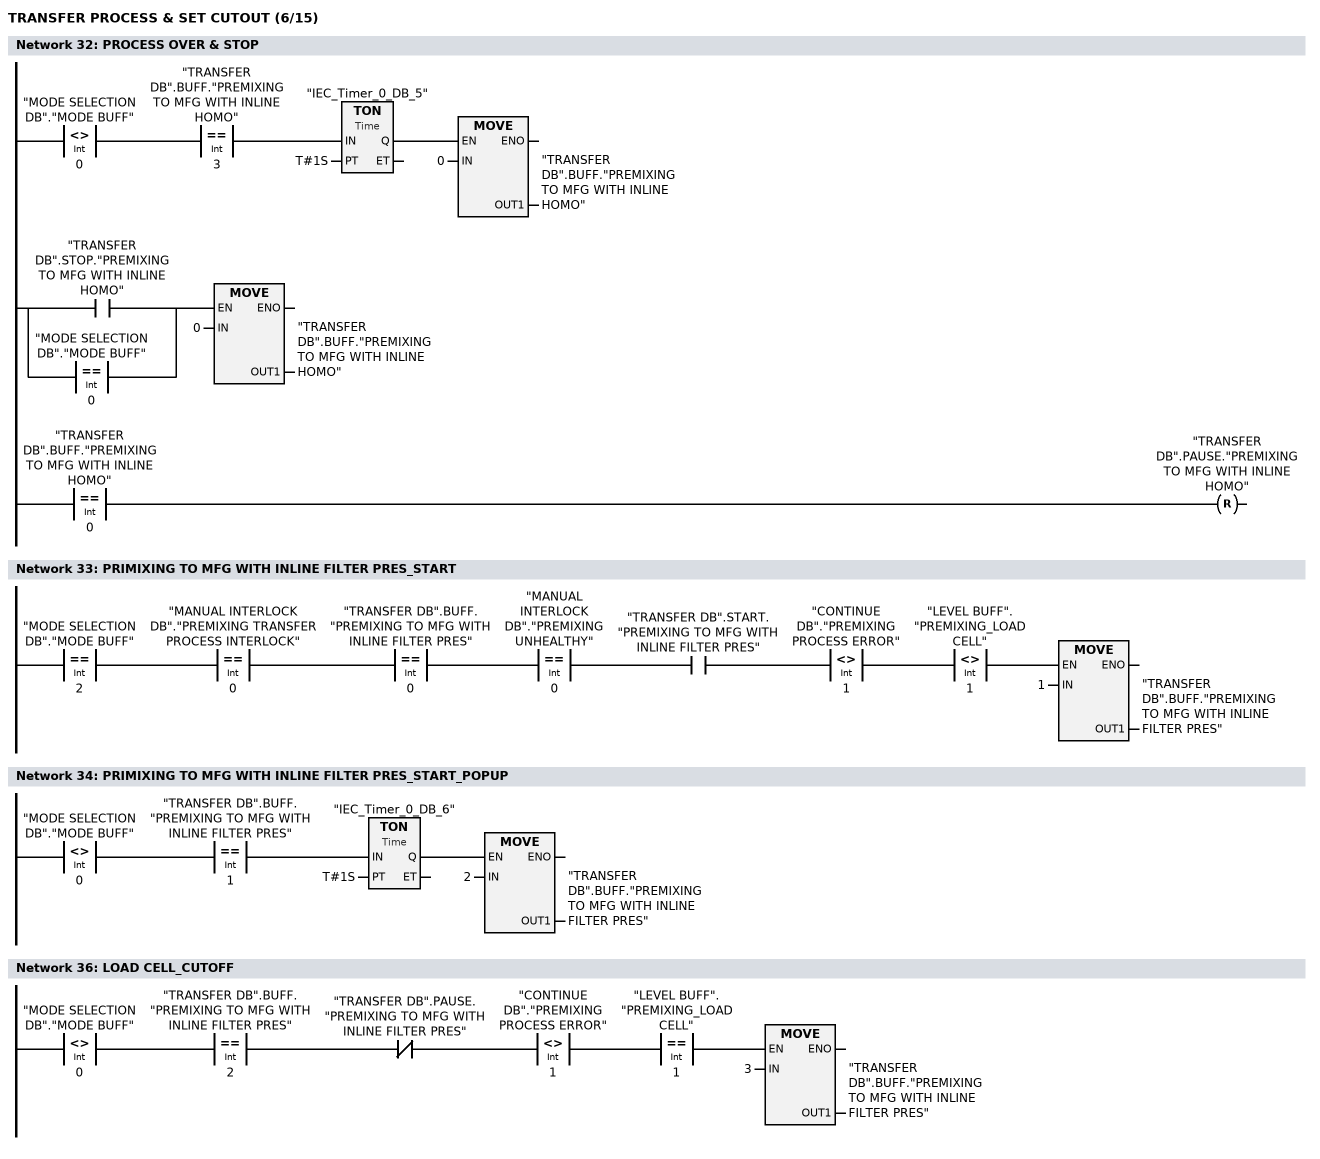
   RUNG wire#powerrail
      { S7_Templates := "SrcType := Int" } NE_Contact(in1 := "MODE SELECTION DB"."MODE BUFF", in2 := 0)
      { S7_Templates := "SrcType := Int" } EQ_Contact(in1 := "TRANSFER DB".BUFF."PREMIXING TO MFG WITH INLINE HOMO", in2 := 3)
      { S7_Templates := "time_type := Time" } "IEC_Timer_0_DB_5".TON(pt := T#1S, et =>)
      Move(in := 0, out1 => "TRANSFER DB".BUFF."PREMIXING TO MFG WITH INLINE HOMO")
   END_RUNG
   RUNG wire#powerrail
      Contact( "TRANSFER DB".STOP."PREMIXING TO MFG WITH INLINE HOMO" )
      wire#w1
      Move(in := 0, out1 => "TRANSFER DB".BUFF."PREMIXING TO MFG WITH INLINE HOMO")
   END_RUNG
   RUNG wire#powerrail
      { S7_Templates := "SrcType := Int" } EQ_Contact(in1 := "MODE SELECTION DB"."MODE BUFF", in2 := 0)
   END_RUNG wire#w1
   RUNG wire#powerrail
      { S7_Templates := "SrcType := Int" } EQ_Contact(in1 := "TRANSFER DB".BUFF."PREMIXING TO MFG WITH INLINE HOMO", in2 := 0)
      R_Coil( "TRANSFER DB".PAUSE."PREMIXING TO MFG WITH INLINE HOMO" )
   END_RUNG
   // the same network as SCL:
   "IEC_Timer_0_DB_5".TON(IN := ("MODE SELECTION DB"."MODE BUFF" <> 0) AND ("TRANSFER DB".BUFF."PREMIXING TO MFG WITH INLINE HOMO" = 3),
                          PT := T#1S);
   IF "IEC_Timer_0_DB_5".Q THEN "TRANSFER DB".BUFF."PREMIXING TO MFG WITH INLINE HOMO" := 0; END_IF;
   IF "TRANSFER DB".STOP."PREMIXING TO MFG WITH INLINE HOMO" OR ("MODE SELECTION DB"."MODE BUFF" = 0) THEN
       "TRANSFER DB".BUFF."PREMIXING TO MFG WITH INLINE HOMO" := 0;
   END_IF;
   IF "TRANSFER DB".BUFF."PREMIXING TO MFG WITH INLINE HOMO" = 0 THEN
       "TRANSFER DB".PAUSE."PREMIXING TO MFG WITH INLINE HOMO" := FALSE;
   END_IF;
END_REGION

REGION Network 33: PRIMIXING TO MFG WITH INLINE FILTER PRES_START
   RUNG wire#powerrail
      { S7_Templates := "SrcType := Int" } EQ_Contact(in1 := "MODE SELECTION DB"."MODE BUFF", in2 := 2)
      { S7_Templates := "SrcType := Int" } EQ_Contact(in1 := "MANUAL INTERLOCK DB"."PREMIXING TRANSFER PROCESS INTERLOCK", in2 := 0)
      { S7_Templates := "SrcType := Int" } EQ_Contact(in1 := "TRANSFER DB".BUFF."PREMIXING TO MFG WITH INLINE FILTER PRES", in2 := 0)
      { S7_Templates := "SrcType := Int" } EQ_Contact(in1 := "MANUAL INTERLOCK DB"."PREMIXING UNHEALTHY", in2 := 0)
      Contact( "TRANSFER DB".START."PREMIXING TO MFG WITH INLINE FILTER PRES" )
      { S7_Templates := "SrcType := Int" } NE_Contact(in1 := "CONTINUE DB"."PREMIXING PROCESS ERROR", in2 := 1)
      { S7_Templates := "SrcType := Int" } NE_Contact(in1 := "LEVEL BUFF"."PREMIXING_LOAD CELL", in2 := 1)
      Move(in := 1, out1 => "TRANSFER DB".BUFF."PREMIXING TO MFG WITH INLINE FILTER PRES")
   END_RUNG
   // the same network as SCL:
   IF ("MODE SELECTION DB"."MODE BUFF" = 2) AND ("MANUAL INTERLOCK DB"."PREMIXING TRANSFER PROCESS INTERLOCK" = 0) AND ("TRANSFER DB".BUFF."PREMIXING TO MFG WITH INLINE FILTER PRES" = 0) AND ("MANUAL INTERLOCK DB"."PREMIXING UNHEALTHY" = 0) AND "TRANSFER DB".START."PREMIXING TO MFG WITH INLINE FILTER PRES" AND ("CONTINUE DB"."PREMIXING PROCESS ERROR" <> 1) AND ("LEVEL BUFF"."PREMIXING_LOAD CELL" <> 1) THEN
       "TRANSFER DB".BUFF."PREMIXING TO MFG WITH INLINE FILTER PRES" := 1;
   END_IF;
END_REGION

REGION Network 34: PRIMIXING TO MFG WITH INLINE FILTER PRES_START_POPUP
   RUNG wire#powerrail
      { S7_Templates := "SrcType := Int" } NE_Contact(in1 := "MODE SELECTION DB"."MODE BUFF", in2 := 0)
      { S7_Templates := "SrcType := Int" } EQ_Contact(in1 := "TRANSFER DB".BUFF."PREMIXING TO MFG WITH INLINE FILTER PRES", in2 := 1)
      { S7_Templates := "time_type := Time" } "IEC_Timer_0_DB_6".TON(pt := T#1S, et =>)
      Move(in := 2, out1 => "TRANSFER DB".BUFF."PREMIXING TO MFG WITH INLINE FILTER PRES")
   END_RUNG
   // the same network as SCL:
   "IEC_Timer_0_DB_6".TON(IN := ("MODE SELECTION DB"."MODE BUFF" <> 0) AND ("TRANSFER DB".BUFF."PREMIXING TO MFG WITH INLINE FILTER PRES" = 1),
                          PT := T#1S);
   IF "IEC_Timer_0_DB_6".Q THEN "TRANSFER DB".BUFF."PREMIXING TO MFG WITH INLINE FILTER PRES" := 2; END_IF;
END_REGION

